C05444=1060.033,39.015,-71.744,171.703,28.984,155.388
C05445=1060.027,38.766,-71.728,171.703,28.981,155.388
C05446=1060.021,38.516,-71.712,171.701,28.979,155.387
C05447=1060.015,38.267,-71.695,171.699,28.976,155.387
C05448=1060.009,38.018,-71.679,171.698,28.973,155.387
C05449=1060.003,37.768,-71.663,171.696,28.971,155.386
C05450=1059.997,37.518,-71.646,171.695,28.968,155.386
C05451=1059.991,37.269,-71.630,171.693,28.966,155.386
C05452=1059.985,37.020,-71.614,171.692,28.963,155.385
C05453=1059.979,36.770,-71.598,171.690,28.961,155.385
C05454=1059.973,36.521,-71.583,171.688,28.959,155.385
C05455=1059.967,36.271,-71.566,171.688,28.956,155.384
C05456=1059.961,36.022,-71.550,171.686,28.954,155.384
C05457=1059.955,35.773,-71.534,171.684,28.951,155.383
C05458=1059.949,35.523,-71.518,171.683,28.949,155.383
C05459=1059.942,35.274,-71.502,171.681,28.946,155.383
C05460=1059.936,35.024,-71.485,171.680,28.944,155.382
C05461=1059.930,34.775,-71.469,171.679,28.941,155.382
C05462=1059.924,34.526,-71.453,171.677,28.939,155.382
C05463=1059.918,34.276,-71.437,171.675,28.936,155.381
C05464=1059.911,34.027,-71.422,171.674,28.933,155.381
C05465=1059.905,33.777,-71.405,171.673,28.931,155.381
C05466=1059.900,33.528,-71.389,171.671,28.929,155.380
C05467=1059.894,33.278,-71.373,171.670,28.927,155.380
C05468=1059.888,33.029,-71.357,171.668,28.924,155.380
C05469=1059.881,32.779,-71.342,171.666,28.922,155.379
C05470=1059.875,32.530,-71.325,171.666,28.919,155.379
C05471=1059.869,32.281,-71.309,171.664,28.916,155.379
C05472=1059.863,32.031,-71.293,171.662,28.914,155.378
C05473=1059.857,31.782,-71.277,171.661,28.911,155.378
C05474=1059.851,31.532,-71.262,171.659,28.909,155.378
C05475=1059.845,31.283,-71.245,171.658,28.906,155.377
C05476=1059.839,31.034,-71.229,171.657,28.904,155.377
C05477=1059.832,30.785,-71.213,171.655,28.901,155.377
C05478=1059.827,30.535,-71.198,171.653,28.899,155.376
C05479=1059.820,30.251,-71.179,171.652,28.896,155.376
C05480=1059.813,29.965,-71.162,171.650,28.893,155.375
C05481=1059.806,29.681,-71.143,171.649,28.890,155.375
C05482=1059.799,29.396,-71.125,171.647,28.888,155.375
C05483=1059.794,29.146,-71.108,171.645,28.885,155.374
C05484=1059.787,28.897,-71.093,171.644,28.883,155.374
C05485=1059.781,28.647,-71.077,171.642,28.880,155.374
C05486=1059.775,28.398,-71.061,171.641,28.878,155.373
C05487=1059.769,28.148,-71.046,171.640,28.876,155.373
C05488=1059.763,27.899,-71.030,171.638,28.873,155.373
C05489=1059.756,27.650,-71.014,171.636,28.871,155.372
C05490=1059.751,27.400,-70.999,171.635,28.868,155.372
C05491=1059.745,27.151,-70.982,171.634,28.866,155.372
C05492=1059.738,26.901,-70.967,171.632,28.863,155.371
C05493=1059.732,26.652,-70.951,171.631,28.861,155.371
C05494=1059.726,26.402,-70.935,171.629,28.858,155.371
C05495=1059.721,26.153,-70.920,171.627,28.856,155.370
C05496=1059.714,25.904,-70.905,171.626,28.853,155.370
C05497=1059.708,25.654,-70.889,171.625,28.851,155.370
C05498=1059.702,25.405,-70.873,171.623,28.848,155.369
C05499=1059.696,25.156,-70.857,171.622,28.846,155.369
C05500=1059.690,24.906,-70.842,171.620,28.843,155.368
C05501=1059.683,24.657,-70.826,171.618,28.841,155.368
C05502=1059.678,24.407,-70.810,171.618,28.838,155.368
C05503=1059.671,24.158,-70.795,171.616,28.836,155.367
C05504=1059.665,23.908,-70.779,171.614,28.833,155.367
C05505=1059.659,23.659,-70.764,171.613,28.831,155.367
C05506=1059.653,23.409,-70.748,171.611,28.829,155.367
C05507=1059.646,23.160,-70.732,171.609,28.826,155.366
C05508=1059.641,22.910,-70.717,171.608,28.824,155.366
C05509=1059.634,22.661,-70.702,171.607,28.822,155.365
C05510=1059.629,22.412,-70.686,171.605,28.819,155.365
C05511=1059.622,22.162,-70.670,171.604,28.817,155.365
C05512=1059.617,21.913,-70.655,171.602,28.814,155.365
C05513=1059.610,21.663,-70.639,171.601,28.812,155.364
C05514=1059.604,21.414,-70.624,171.599,28.810,155.364
C05515=1059.598,21.164,-70.607,171.598,28.807,155.363
C05516=1059.592,20.914,-70.592,171.596,28.805,155.363
C05517=1059.587,20.665,-70.577,171.595,28.802,155.363
C05518=1059.580,20.416,-70.562,171.593,28.800,155.362
C05519=1059.574,20.166,-70.546,171.592,28.797,155.362
C05520=1059.568,19.917,-70.530,171.590,28.795,155.362
C05521=1059.561,19.668,-70.515,171.589,28.793,155.362
C05522=1059.556,19.418,-70.500,171.587,28.790,155.361
C05523=1059.549,19.169,-70.484,171.585,28.788,155.361
C05524=1059.543,18.920,-70.470,171.584,28.785,155.360
C05525=1059.538,18.670,-70.454,171.583,28.783,155.360
C05526=1059.531,18.421,-70.438,171.581,28.781,155.360
C05527=1059.525,18.171,-70.423,171.580,28.778,155.359
C05528=1059.519,17.921,-70.408,171.578,28.776,155.359
C05529=1059.512,17.672,-70.392,171.577,28.773,155.359
C05530=1059.507,17.423,-70.377,171.576,28.771,155.359
C05531=1059.501,17.173,-70.362,171.574,28.769,155.358
C05532=1059.494,16.924,-70.346,171.572,28.766,155.358
C05533=1059.488,16.674,-70.331,171.571,28.764,155.358
C05534=1059.482,16.424,-70.316,171.569,28.761,155.357
C05535=1059.477,16.176,-70.300,171.567,28.759,155.357
C05536=1059.470,15.926,-70.285,171.567,28.757,155.357
C05537=1059.464,15.676,-70.270,171.565,28.754,155.356
C05538=1059.458,15.426,-70.255,171.563,28.752,155.356
C05539=1059.452,15.177,-70.239,171.562,28.749,155.356
C05540=1059.446,14.928,-70.224,171.560,28.747,155.355
C05541=1059.440,14.678,-70.209,171.558,28.744,155.355
C05542=1059.434,14.429,-70.194,171.558,28.742,155.355
C05543=1059.427,14.146,-70.176,171.555,28.739,155.354
C05544=1059.419,13.861,-70.160,171.554,28.737,155.354
C05545=1059.412,13.579,-70.142,171.552,28.734,155.354
C05546=1059.405,13.295,-70.125,171.550,28.731,155.353
C05547=1059.399,13.046,-70.110,171.549,28.729,155.353
C05548=1059.393,12.796,-70.095,171.547,28.727,155.353
C05549=1059.386,12.546,-70.080,171.546,28.725,155.352
C05550=1059.381,12.297,-70.065,171.545,28.722,155.352
C05551=1059.375,12.048,-70.050,171.543,28.720,155.352
C05552=1059.369,11.798,-70.035,171.541,28.717,155.351
C05553=1059.362,11.549,-70.019,171.540,28.715,155.351
C05554=1059.356,11.300,-70.005,171.538,28.712,155.351
C05555=1059.350,11.050,-69.990,171.537,28.710,155.350
C05556=1059.343,10.801,-69.975,171.536,28.708,155.350
C05557=1059.337,10.551,-69.960,171.534,28.705,155.350
C05558=1059.331,10.301,-69.945,171.532,28.703,155.349
C05559=1059.325,10.052,-69.930,171.531,28.701,155.349
C05560=1059.319,9.802,-69.915,171.529,28.699,155.349
C05561=1059.313,9.553,-69.900,171.527,28.696,155.349
C05562=1059.306,9.303,-69.885,171.527,28.694,155.348
C05563=1059.301,9.054,-69.870,171.525,28.692,155.348
C05564=1059.294,8.804,-69.855,171.523,28.689,155.348
C05565=1059.288,8.555,-69.840,171.522,28.687,155.347
C05566=1059.282,8.306,-69.826,171.520,28.684,155.347
C05567=1059.276,8.056,-69.811,171.518,28.682,155.347
C05568=1059.269,7.806,-69.796,171.516,28.680,155.347
C05569=1059.264,7.556,-69.780,171.516,28.677,155.346
C05570=1059.258,7.308,-69.766,171.514,28.675,155.346
C05571=1059.251,7.058,-69.751,171.512,28.673,155.346
C05572=1059.245,6.808,-69.736,171.511,28.671,155.345
C05573=1059.239,6.559,-69.721,171.509,28.668,155.345
C05574=1059.233,6.310,-69.706,171.507,28.666,155.345
C05575=1059.226,6.060,-69.691,171.506,28.664,155.344
C05576=1059.221,5.811,-69.677,171.505,28.662,155.344
C05577=1059.214,5.561,-69.662,171.503,28.659,155.344
C05578=1059.208,5.312,-69.647,171.502,28.656,155.343
C05579=1059.202,5.063,-69.632,171.500,28.654,155.343
C05580=1059.196,4.813,-69.617,171.498,28.652,155.343
C05581=1059.189,4.563,-69.602,171.497,28.649,155.342
C05582=1059.184,4.314,-69.588,171.495,28.647,155.342
C05583=1059.178,4.064,-69.573,171.494,28.645,155.342
C05584=1059.172,3.814,-69.558,171.493,28.643,155.342
C05585=1059.166,3.565,-69.544,171.491,28.640,155.341
C05586=1059.160,3.316,-69.529,171.489,28.638,155.341
C05587=1059.153,3.066,-69.514,171.488,28.636,155.341
C05588=1059.148,2.817,-69.499,171.486,28.633,155.340
C05589=1059.141,2.567,-69.484,171.484,28.631,155.340
C05590=1059.136,2.318,-69.470,171.484,28.629,155.340
C05591=1059.129,2.068,-69.455,171.482,28.626,155.339
C05592=1059.123,1.818,-69.440,171.480,28.624,155.339
C05593=1059.117,1.569,-69.426,171.479,28.621,155.339
C05594=1059.111,1.320,-69.411,171.477,28.619,155.338
C05595=1059.105,1.070,-69.397,171.475,28.617,155.338
C05596=1059.099,0.821,-69.382,171.474,28.615,155.338
C05597=1059.093,0.572,-69.367,171.473,28.612,155.338
C05598=1059.087,0.322,-69.353,171.471,28.610,155.337
C05599=1059.080,0.072,-69.338,171.470,28.608,155.337
C05600=1059.075,-0.177,-69.324,171.468,28.605,155.337
C05601=1059.068,-0.427,-69.309,171.466,28.603,155.336
C05602=1059.063,-0.676,-69.294,171.465,28.600,155.336
C05603=1059.056,-0.926,-69.279,171.463,28.598,155.336
C05604=1059.051,-1.175,-69.265,171.461,28.596,155.336
C05605=1059.044,-1.425,-69.250,171.461,28.593,155.335
C05606=1059.039,-1.674,-69.236,171.459,28.591,155.335
C05607=1059.032,-1.956,-69.219,171.457,28.589,155.335
C05608=1059.025,-2.237,-69.203,171.455,28.586,155.334
C05609=1059.018,-2.519,-69.187,171.453,28.583,155.334
C05610=1059.012,-2.801,-69.170,171.452,28.581,155.334
C05611=1059.006,-3.050,-69.155,171.450,28.578,155.333
C05612=1059.000,-3.299,-69.141,171.449,28.576,155.333
C05613=1058.993,-3.549,-69.127,171.448,28.574,155.333
C05614=1058.987,-3.798,-69.113,171.446,28.572,155.332
C05615=1058.981,-4.048,-69.098,171.444,28.569,155.332
C05616=1058.975,-4.298,-69.083,171.443,28.567,155.332
C05617=1058.968,-4.547,-69.069,171.441,28.565,155.331
C05618=1058.962,-4.797,-69.055,171.439,28.563,155.331
C05619=1058.956,-5.046,-69.041,171.438,28.560,155.331
C05620=1058.950,-5.296,-69.027,171.436,28.558,155.331
C05621=1058.944,-5.545,-69.012,171.435,28.556,155.330
C05622=1058.937,-5.794,-68.997,171.433,28.554,155.330
C05623=1058.932,-6.044,-68.984,171.432,28.552,155.330
C05624=1058.925,-6.293,-68.969,171.430,28.550,155.330
C05625=1058.919,-6.543,-68.955,171.428,28.547,155.329
C05626=1058.913,-6.793,-68.940,171.427,28.545,155.329
C05627=1058.906,-7.043,-68.927,171.425,28.543,155.329
C05628=1058.900,-7.291,-68.912,171.424,28.540,155.328
C05629=1058.894,-7.542,-68.898,171.422,28.538,155.328
C05630=1058.888,-7.790,-68.884,171.420,28.536,155.328
C05631=1058.882,-8.041,-68.870,171.419,28.534,155.328
C05632=1058.876,-8.290,-68.855,171.418,28.531,155.327
C05633=1058.870,-8.540,-68.841,171.416,28.529,155.327
C05634=1058.863,-8.789,-68.827,171.414,28.527,155.327
C05635=1058.858,-9.038,-68.813,171.413,28.525,155.326
C05636=1058.851,-9.288,-68.798,171.411,28.522,155.326
C05637=1058.845,-9.537,-68.785,171.409,28.520,155.326
C05638=1058.839,-9.787,-68.770,171.408,28.518,155.326
C05639=1058.833,-10.036,-68.756,171.406,28.516,155.325
C05640=1058.827,-10.286,-68.742,171.405,28.514,155.325
C05641=1058.821,-10.535,-68.728,171.404,28.512,155.325
C05642=1058.815,-10.786,-68.714,171.402,28.509,155.325
C05643=1058.808,-11.034,-68.700,171.400,28.507,155.324
C05644=1058.802,-11.284,-68.685,171.399,28.505,155.324
C05645=1058.797,-11.534,-68.672,171.397,28.503,155.324
C05646=1058.790,-11.783,-68.658,171.395,28.500,155.323
C05647=1058.784,-12.033,-68.643,171.394,28.498,155.323
C05648=1058.779,-12.282,-68.630,171.392,28.496,155.323
C05649=1058.771,-12.532,-68.615,171.390,28.494,155.323
C05650=1058.766,-12.781,-68.601,171.389,28.492,155.322
C05651=1058.760,-13.031,-68.588,171.388,28.490,155.322
C05652=1058.753,-13.280,-68.573,171.386,28.487,155.322
C05653=1058.748,-13.530,-68.559,171.385,28.485,155.322
C05654=1058.741,-13.780,-68.546,171.383,28.483,155.321
C05655=1058.735,-14.029,-68.531,171.381,28.481,155.321
C05656=1058.730,-14.278,-68.517,171.380,28.478,155.321
C05657=1058.723,-14.528,-68.504,171.378,28.476,155.320
C05658=1058.717,-14.777,-68.489,171.376,28.474,155.320
C05659=1058.711,-15.027,-68.476,171.375,28.472,155.320
C05660=1058.705,-15.277,-68.461,171.373,28.469,155.320
C05661=1058.699,-15.526,-68.448,171.371,28.467,155.319
C05662=1058.692,-15.776,-68.433,171.371,28.465,155.319
C05663=1058.686,-16.025,-68.420,171.369,28.464,155.319
C05664=1058.681,-16.275,-68.406,171.367,28.461,155.319
C05665=1058.674,-16.525,-68.392,171.365,28.459,155.318
C05666=1058.668,-16.774,-68.379,171.364,28.457,155.318
C05667=1058.661,-17.024,-68.364,171.362,28.455,155.318
C05668=1058.655,-17.273,-68.351,171.360,28.452,155.318
C05669=1058.650,-17.522,-68.337,171.359,28.450,155.317
C05670=1058.643,-17.772,-68.323,171.357,28.449,155.317
C05671=1058.636,-18.052,-68.307,171.355,28.446,155.317
C05672=1058.629,-18.332,-68.293,171.354,28.443,155.316
C05673=1058.622,-18.612,-68.277,171.352,28.441,155.316
C05674=1058.615,-18.892,-68.262,171.350,28.439,155.316
C05675=1058.609,-19.141,-68.248,171.349,28.437,155.316
C05676=1058.603,-19.391,-68.234,171.347,28.435,155.315
C05677=1058.596,-19.640,-68.220,171.345,28.432,155.315
C05678=1058.590,-19.889,-68.207,171.344,28.430,155.315
C05679=1058.584,-20.140,-68.193,171.342,28.428,155.315
C05680=1058.578,-20.389,-68.179,171.340,28.426,155.314
C05681=1058.573,-20.639,-68.166,171.339,28.424,155.314
C05682=1058.566,-20.889,-68.152,171.337,28.422,155.314
C05683=1058.559,-21.138,-68.139,171.335,28.419,155.314
C05684=1058.554,-21.387,-68.125,171.334,28.418,155.314
C05685=1058.548,-21.637,-68.112,171.332,28.416,155.313
C05686=1058.542,-21.887,-68.097,171.330,28.413,155.313
C05687=1058.535,-22.136,-68.084,171.329,28.411,155.313
C05688=1058.529,-22.385,-68.071,171.328,28.409,155.312
C05689=1058.523,-22.636,-68.057,171.326,28.407,155.312
C05690=1058.517,-22.885,-68.043,171.324,28.405,155.312
C05691=1058.511,-23.134,-68.030,171.323,28.403,155.312
C05692=1058.505,-23.384,-68.016,171.321,28.401,155.311
C05693=1058.498,-23.634,-68.003,171.319,28.399,155.311
C05694=1058.492,-23.883,-67.989,171.318,28.396,155.311
C05695=1058.487,-24.133,-67.975,171.316,28.395,155.311
C05696=1058.481,-24.382,-67.962,171.314,28.392,155.310
C05697=1058.474,-24.632,-67.948,171.313,28.390,155.310
C05698=1058.468,-24.881,-67.935,171.311,28.388,155.310
C05699=1058.462,-25.131,-67.921,171.309,28.386,155.310
C05700=1058.456,-25.380,-67.908,171.308,28.384,155.310
C05701=1058.450,-25.630,-67.894,171.306,28.382,155.309
C05702=1058.444,-25.880,-67.881,171.304,28.380,155.309
C05703=1058.437,-26.129,-67.867,171.303,28.377,155.309
C05704=1058.432,-26.378,-67.853,171.301,28.376,155.309
C05705=1058.426,-26.628,-67.840,171.300,28.374,155.308
C05706=1058.419,-26.878,-67.827,171.299,28.371,155.308
C05707=1058.414,-27.128,-67.813,171.297,28.369,155.308
C05708=1058.407,-27.377,-67.800,171.295,28.368,155.308
C05709=1058.401,-27.626,-67.787,171.294,28.365,155.307
C05710=1058.394,-27.876,-67.773,171.292,28.364,155.307
C05711=1058.388,-28.126,-67.760,171.290,28.361,155.307
C05712=1058.382,-28.375,-67.747,171.288,28.359,155.307
C05713=1058.376,-28.625,-67.734,171.287,28.358,155.306
C05714=1058.369,-28.875,-67.720,171.285,28.355,155.306
C05715=1058.363,-29.124,-67.707,171.283,28.353,155.306
C05716=1058.358,-29.373,-67.693,171.282,28.351,155.306
C05717=1058.351,-29.623,-67.680,171.280,28.349,155.306
C05718=1058.345,-29.873,-67.668,171.278,28.348,155.305
C05719=1058.339,-30.123,-67.654,171.277,28.345,155.305
C05720=1058.332,-30.372,-67.641,171.275,28.343,155.305
C05721=1058.326,-30.621,-67.627,171.273,28.341,155.305
C05722=1058.320,-30.870,-67.614,171.272,28.339,155.304
C05723=1058.314,-31.120,-67.602,171.270,28.337,155.304
C05724=1058.308,-31.370,-67.588,171.268,28.335,155.304
C05725=1058.301,-31.619,-67.575,171.266,28.333,155.304
C05726=1058.296,-31.870,-67.561,171.265,28.331,155.304
C05727=1058.290,-32.119,-67.548,171.263,28.329,155.303
C05728=1058.283,-32.368,-67.535,171.261,28.327,155.303
C05729=1058.277,-32.617,-67.522,171.260,28.325,155.303
C05730=1058.271,-32.867,-67.509,171.259,28.323,155.303
C05731=1058.265,-33.117,-67.495,171.257,28.322,155.302
C05732=1058.258,-33.367,-67.482,171.256,28.319,155.302
C05733=1058.252,-33.616,-67.470,171.254,28.318,155.302
C05734=1058.246,-33.866,-67.456,171.252,28.315,155.302
C05735=1058.240,-34.145,-67.442,171.250,28.313,155.302
C05736=1058.233,-34.424,-67.427,171.248,28.311,155.301
C05737=1058.226,-34.703,-67.413,171.246,28.308,155.301
C05738=1058.218,-34.982,-67.398,171.245,28.307,155.301
C05739=1058.212,-35.232,-67.385,171.243,28.305,155.301
C05740=1058.206,-35.482,-67.372,171.241,28.302,155.300
C05741=1058.200,-35.731,-67.359,171.239,28.301,155.300
C05742=1058.194,-35.981,-67.346,171.238,28.298,155.300
C05743=1058.188,-36.230,-67.333,171.236,28.297,155.300
C05744=1058.182,-36.480,-67.320,171.234,28.295,155.300
C05745=1058.177,-36.729,-67.306,171.233,28.293,155.299
C05746=1058.171,-36.979,-67.294,171.231,28.291,155.299
C05747=1058.164,-37.229,-67.280,171.229,28.289,155.299
C05748=1058.159,-37.478,-67.268,171.228,28.287,155.299
C05749=1058.152,-37.728,-67.255,171.226,28.285,155.298
C05750=1058.146,-37.978,-67.242,171.224,28.283,155.298
C05751=1058.140,-38.227,-67.229,171.223,28.281,155.298
C05752=1058.134,-38.477,-67.216,171.221,28.279,155.298
C05753=1058.128,-38.726,-67.203,171.219,28.277,155.298
C05754=1058.121,-38.976,-67.191,171.217,28.275,155.297
C05755=1058.115,-39.226,-67.177,171.216,28.273,155.297
C05756=1058.109,-39.475,-67.165,171.214,28.271,155.297
C05757=1058.102,-39.725,-67.152,171.212,28.270,155.297
C05758=1058.097,-39.975,-67.139,171.211,28.267,155.297
C05759=1058.090,-40.224,-67.126,171.209,28.266,155.296
C05760=1058.084,-40.473,-67.114,171.207,28.264,155.296
C05761=1058.077,-40.723,-67.100,171.206,28.262,155.296
C05762=1058.072,-40.973,-67.088,171.204,28.260,155.296
C05763=1058.066,-41.222,-67.075,171.202,28.258,155.296
C05764=1058.059,-41.472,-67.062,171.200,28.256,155.295
C05765=1058.053,-41.721,-67.050,171.199,28.254,155.295
C05766=1058.047,-41.970,-67.037,171.197,28.253,155.295
C05767=1058.041,-42.220,-67.024,171.195,28.251,155.295
C05768=1058.035,-42.470,-67.012,171.194,28.249,155.295
C05769=1058.029,-42.720,-66.998,171.192,28.247,155.295
C05770=1058.022,-42.969,-66.987,171.190,28.245,155.294
C05771=1058.016,-43.219,-66.974,171.188,28.243,155.294
C05772=1058.010,-43.468,-66.961,171.187,28.241,155.294
C05773=1058.004,-43.718,-66.948,171.185,28.239,155.294
C05774=1057.998,-43.968,-66.936,171.183,28.238,155.294
C05775=1057.991,-44.217,-66.923,171.182,28.236,155.293
C05776=1057.985,-44.467,-66.910,171.180,28.234,155.293
C05777=1057.979,-44.717,-66.898,171.178,28.232,155.293
C05778=1057.973,-44.966,-66.885,171.176,28.230,155.293
C05779=1057.966,-45.216,-66.873,171.175,28.228,155.293
C05780=1057.960,-45.465,-66.860,171.173,28.227,155.293
C05781=1057.955,-45.715,-66.847,171.171,28.225,155.292
C05782=1057.948,-45.965,-66.834,171.170,28.223,155.292
C05783=1057.942,-46.214,-66.822,171.168,28.221,155.292
C05784=1057.936,-46.464,-66.810,171.166,28.219,155.292
C05785=1057.930,-46.714,-66.797,171.165,28.217,155.292
C05786=1057.924,-46.963,-66.784,171.163,28.216,155.291
C05787=1057.917,-47.213,-66.772,171.161,28.214,155.291
C05788=1057.911,-47.463,-66.759,171.159,28.212,155.291
C05789=1057.906,-47.712,-66.747,171.158,28.210,155.291
C05790=1057.900,-47.961,-66.734,171.156,28.208,155.291
C05791=1057.893,-48.211,-66.722,171.154,28.207,155.291
C05792=1057.887,-48.461,-66.709,171.153,28.204,155.290
C05793=1057.881,-48.710,-66.697,171.151,28.203,155.290
C05794=1057.875,-48.960,-66.684,171.149,28.201,155.290
C05795=1057.869,-49.210,-66.672,171.147,28.199,155.290
C05796=1057.862,-49.459,-66.659,171.146,28.197,155.290
C05797=1057.856,-49.709,-66.646,171.144,28.196,155.289
C05798=1057.851,-49.958,-66.634,171.142,28.194,155.289
C05799=1057.843,-50.238,-66.620,171.141,28.192,155.289
C05800=1057.836,-50.518,-66.607,171.139,28.190,155.289
C05801=1057.830,-50.797,-66.593,171.136,28.187,155.289
C05802=1057.823,-51.077,-66.579,171.134,28.186,155.289
C05803=1057.816,-51.326,-66.568,171.133,28.184,155.288
C05804=1057.810,-51.576,-66.555,171.131,28.182,155.288
C05805=1057.804,-51.825,-66.542,171.129,28.181,155.288
C05806=1057.798,-52.075,-66.530,171.128,28.179,155.288
C05807=1057.791,-52.325,-66.518,171.126,28.178,155.288
C05808=1057.784,-52.574,-66.506,171.124,28.176,155.288
C05809=1057.778,-52.824,-66.493,171.122,28.174,155.287
C05810=1057.772,-53.074,-66.481,171.121,28.173,155.287
C05811=1057.766,-53.323,-66.469,171.119,28.171,155.287
C05812=1057.759,-53.573,-66.457,171.117,28.169,155.287
C05813=1057.753,-53.822,-66.445,171.115,28.168,155.287
C05814=1057.747,-54.072,-66.433,171.114,28.166,155.287
C05815=1057.741,-54.321,-66.421,171.112,28.164,155.287
C05816=1057.735,-54.571,-66.408,171.110,28.163,155.286
C05817=1057.728,-54.821,-66.396,171.109,28.161,155.286
C05818=1057.721,-55.070,-66.384,171.107,28.159,155.286
C05819=1057.716,-55.320,-66.372,171.105,28.158,155.286
C05820=1057.710,-55.570,-66.361,171.103,28.156,155.286
C05821=1057.704,-55.820,-66.348,171.102,28.154,155.286
C05822=1057.697,-56.069,-66.336,171.099,28.152,155.286
C05823=1057.691,-56.319,-66.324,171.097,28.151,155.285
C05824=1057.685,-56.569,-66.312,171.095,28.149,155.285
C05825=1057.678,-56.818,-66.300,171.094,28.147,155.285
C05826=1057.671,-57.068,-66.288,171.092,28.146,155.285
C05827=1057.666,-57.317,-66.276,171.090,28.144,155.285
C05828=1057.659,-57.567,-66.264,171.089,28.142,155.285
C05829=1057.654,-57.816,-66.251,171.087,28.141,155.285
C05830=1057.647,-58.067,-66.240,171.085,28.139,155.284
C05831=1057.641,-58.316,-66.228,171.083,28.137,155.284
C05832=1057.635,-58.565,-66.216,171.082,28.136,155.284
C05833=1057.629,-58.815,-66.204,171.080,28.134,155.284
C05834=1057.622,-59.065,-66.192,171.078,28.132,155.284
C05835=1057.616,-59.314,-66.179,171.076,28.131,155.284
C05836=1057.610,-59.564,-66.168,171.075,28.130,155.284
C05837=1057.604,-59.814,-66.156,171.073,28.128,155.284
C05838=1057.598,-60.063,-66.144,171.071,28.126,155.283
C05839=1057.591,-60.313,-66.132,171.069,28.125,155.283
C05840=1057.584,-60.563,-66.120,171.068,28.123,155.283
C05841=1057.579,-60.812,-66.109,171.066,28.121,155.283
C05842=1057.573,-61.062,-66.097,171.064,28.120,155.283
C05843=1057.566,-61.311,-66.085,171.062,28.118,155.283
C05844=1057.561,-61.561,-66.072,171.061,28.116,155.282
C05845=1057.554,-61.811,-66.061,171.059,28.115,155.282
C05846=1057.548,-62.060,-66.049,171.056,28.113,155.282
C05847=1057.542,-62.310,-66.037,171.055,28.112,155.282
C05848=1057.536,-62.559,-66.025,171.053,28.110,155.282
C05849=1057.530,-62.809,-66.014,171.051,28.108,155.282
C05850=1057.524,-63.059,-66.001,171.049,28.107,155.282
C05851=1057.518,-63.308,-65.990,171.048,28.105,155.282
C05852=1057.511,-63.558,-65.978,171.046,28.103,155.281
C05853=1057.505,-63.808,-65.966,171.044,28.102,155.281
C05854=1057.499,-64.058,-65.954,171.042,28.101,155.281
C05855=1057.493,-64.307,-65.942,171.041,28.099,155.281
C05856=1057.486,-64.557,-65.931,171.039,28.097,155.281
C05857=1057.480,-64.807,-65.919,171.037,28.096,155.281
C05858=1057.475,-65.056,-65.908,171.035,28.094,155.281
C05859=1057.468,-65.306,-65.896,171.034,28.092,155.281
C05860=1057.462,-65.556,-65.883,171.032,28.091,155.281
C05861=1057.456,-65.805,-65.872,171.030,28.090,155.280
C05862=1057.450,-66.055,-65.860,171.028,28.088,155.280
C05863=1057.440,-66.445,-65.842,171.025,28.085,155.280
C05864=1057.431,-66.836,-65.823,171.022,28.083,155.280
C05865=1057.422,-67.226,-65.805,171.020,28.080,155.280
C05866=1057.412,-67.617,-65.787,171.017,28.078,155.280
C05867=1057.406,-67.867,-65.776,171.015,28.077,155.279
C05868=1057.399,-68.116,-65.764,171.014,28.075,155.279
C05869=1057.394,-68.366,-65.752,171.012,28.073,155.279
C05870=1057.388,-68.616,-65.740,171.010,28.072,155.279
C05871=1057.381,-68.866,-65.729,171.008,28.071,155.279
C05872=1057.375,-69.115,-65.717,171.006,28.069,155.279
C05873=1057.370,-69.365,-65.706,171.004,28.067,155.279
C05874=1057.364,-69.614,-65.694,171.002,28.065,155.279
C05875=1057.357,-69.864,-65.683,171.000,28.064,155.278
C05876=1057.351,-70.113,-65.671,170.999,28.063,155.278
C05877=1057.346,-70.364,-65.659,170.997,28.061,155.278
C05878=1057.339,-70.613,-65.647,170.995,28.059,155.278
C05879=1057.333,-70.863,-65.637,170.993,28.058,155.278
C05880=1057.327,-71.112,-65.625,170.992,28.057,155.278
C05881=1057.322,-71.362,-65.613,170.990,28.055,155.278
C05882=1057.315,-71.612,-65.601,170.988,28.053,155.278
C05883=1057.309,-71.861,-65.590,170.986,28.052,155.278
C05884=1057.303,-72.111,-65.579,170.985,28.050,155.277
C05885=1057.297,-72.360,-65.567,170.983,28.049,155.277
C05886=1057.291,-72.611,-65.556,170.981,28.048,155.277
C05887=1057.285,-72.860,-65.544,170.979,28.046,155.277
C05888=1057.279,-73.110,-65.533,170.978,28.044,155.277
C05889=1057.273,-73.359,-65.522,170.975,28.042,155.277
C05890=1057.266,-73.609,-65.510,170.973,28.041,155.277
C05891=1057.261,-73.859,-65.498,170.971,28.040,155.277
C05892=1057.255,-74.108,-65.487,170.970,28.039,155.277
C05893=1057.249,-74.358,-65.476,170.968,28.037,155.276
C05894=1057.243,-74.608,-65.464,170.966,28.035,155.276
C05895=1057.237,-74.857,-65.453,170.964,28.034,155.276
C05896=1057.230,-75.107,-65.442,170.963,28.033,155.276
C05897=1057.224,-75.357,-65.430,170.961,28.031,155.276
C05898=1057.218,-75.607,-65.419,170.959,28.030,155.276
C05899=1057.212,-75.856,-65.407,170.957,28.029,155.276
C05900=1057.206,-76.106,-65.397,170.956,28.027,155.276
C05901=1057.199,-76.356,-65.385,170.954,28.026,155.276
C05902=1057.193,-76.605,-65.374,170.952,28.024,155.276
C05903=1057.186,-76.855,-65.363,170.949,28.023,155.276
C05904=1057.181,-77.104,-65.352,170.947,28.021,155.276
C05905=1057.174,-77.354,-65.341,170.946,28.020,155.275
C05906=1057.168,-77.603,-65.329,170.944,28.019,155.275
C05907=1057.162,-77.853,-65.318,170.942,28.018,155.275
C05908=1057.156,-78.103,-65.307,170.940,28.016,155.275
C05909=1057.150,-78.353,-65.296,170.939,28.015,155.275
C05910=1057.144,-78.603,-65.285,170.937,28.014,155.275
C05911=1057.134,-78.992,-65.268,170.934,28.011,155.275
C05912=1057.125,-79.382,-65.250,170.931,28.009,155.275
C05913=1057.115,-79.771,-65.233,170.928,28.007,155.275
C05914=1057.105,-80.161,-65.215,170.925,28.005,155.275
C05915=1057.100,-80.411,-65.204,170.924,28.004,155.274
C05916=1057.093,-80.661,-65.193,170.922,28.002,155.274
C05917=1057.087,-80.910,-65.183,170.920,28.001,155.274
C05918=1057.080,-81.159,-65.171,170.918,28.000,155.274
C05919=1057.074,-81.409,-65.160,170.915,27.998,155.274
C05920=1057.069,-81.658,-65.149,170.914,27.997,155.274
C05921=1057.062,-81.908,-65.139,170.912,27.996,155.274
C05922=1057.056,-82.158,-65.128,170.910,27.995,155.274
C05923=1057.048,-82.441,-65.116,170.908,27.994,155.274
C05924=1057.041,-82.724,-65.103,170.905,27.992,155.274
C05925=1057.035,-83.007,-65.090,170.904,27.991,155.274
C05926=1057.027,-83.290,-65.078,170.902,27.989,155.274
C05927=1057.021,-83.540,-65.067,170.900,27.988,155.274
C05928=1057.015,-83.789,-65.056,170.897,27.986,155.274
C05929=1057.008,-84.039,-65.045,170.896,27.985,155.274
C05930=1057.003,-84.289,-65.034,170.894,27.984,155.274
C05931=1056.996,-84.539,-65.023,170.892,27.983,155.274
C05932=1056.990,-84.788,-65.013,170.890,27.982,155.274
C05933=1056.984,-85.038,-65.002,170.888,27.981,155.274
C05934=1056.978,-85.288,-64.991,170.887,27.979,155.273
C05935=1056.971,-85.537,-64.980,170.885,27.978,155.273
C05936=1056.965,-85.787,-64.969,170.883,27.977,155.273
C05937=1056.959,-86.037,-64.958,170.881,27.976,155.273
C05938=1056.953,-86.286,-64.948,170.880,27.975,155.273
C05939=1056.947,-86.537,-64.937,170.877,27.973,155.273
C05940=1056.941,-86.786,-64.927,170.875,27.972,155.273
C05941=1056.934,-87.035,-64.916,170.873,27.971,155.273
C05942=1056.928,-87.286,-64.905,170.871,27.970,155.273
C05943=1056.922,-87.535,-64.894,170.870,27.969,155.273
C05944=1056.916,-87.784,-64.884,170.868,27.967,155.273
C05945=1056.909,-88.035,-64.873,170.866,27.966,155.273
C05946=1056.904,-88.284,-64.862,170.864,27.965,155.273
C05947=1056.897,-88.533,-64.851,170.862,27.964,155.273
C05948=1056.891,-88.783,-64.840,170.861,27.963,155.273
C05949=1056.885,-89.033,-64.829,170.858,27.962,155.273
C05950=1056.879,-89.283,-64.820,170.856,27.961,155.273
C05951=1056.873,-89.533,-64.809,170.854,27.959,155.273
C05952=1056.867,-89.782,-64.798,170.852,27.958,155.273
C05953=1056.860,-90.032,-64.787,170.851,27.957,155.273
C05954=1056.854,-90.282,-64.776,170.849,27.956,155.273
C05955=1056.848,-90.531,-64.765,170.847,27.955,155.273
C05956=1056.842,-90.781,-64.756,170.845,27.953,155.273
C05957=1056.836,-91.030,-64.745,170.843,27.952,155.273
C05958=1056.829,-91.280,-64.734,170.842,27.951,155.273
C05959=1056.824,-91.530,-64.723,170.839,27.950,155.273
C05960=1056.818,-91.779,-64.712,170.837,27.949,155.273
C05961=1056.811,-92.030,-64.702,170.835,27.948,155.273
C05962=1056.805,-92.279,-64.692,170.833,27.947,155.272
C05963=1056.800,-92.529,-64.681,170.832,27.945,155.272
C05964=1056.793,-92.778,-64.670,170.830,27.944,155.272
C05965=1056.787,-93.029,-64.660,170.828,27.943,155.272
C05966=1056.781,-93.278,-64.650,170.826,27.942,155.272
C05967=1056.775,-93.527,-64.639,170.824,27.941,155.272
C05968=1056.769,-93.777,-64.628,170.823,27.940,155.272
C05969=1056.762,-94.027,-64.618,170.820,27.938,155.272
C05970=1056.757,-94.277,-64.607,170.818,27.937,155.272
C05971=1056.750,-94.526,-64.597,170.816,27.936,155.272
C05972=1056.745,-94.776,-64.587,170.814,27.935,155.272
C05973=1056.739,-95.026,-64.576,170.813,27.934,155.272
C05974=1056.732,-95.276,-64.565,170.811,27.933,155.272
C05975=1056.726,-95.526,-64.555,170.809,27.932,155.272
C05976=1056.720,-95.775,-64.545,170.807,27.931,155.272
C05977=1056.714,-96.024,-64.534,170.805,27.930,155.272
C05978=1056.709,-96.274,-64.524,170.804,27.929,155.272
C05979=1056.702,-96.524,-64.513,170.801,27.927,155.272
C05980=1056.696,-96.774,-64.502,170.799,27.926,155.272
C05981=1056.690,-97.024,-64.492,170.797,27.925,155.272
C05982=1056.684,-97.273,-64.482,170.795,27.924,155.272
C05983=1056.678,-97.523,-64.472,170.793,27.924,155.272
C05984=1056.672,-97.772,-64.461,170.792,27.923,155.272
C05985=1056.665,-98.022,-64.451,170.790,27.922,155.272
C05986=1056.660,-98.272,-64.440,170.788,27.920,155.272
C05987=1056.652,-98.557,-64.429,170.785,27.919,155.272
C05988=1056.645,-98.843,-64.417,170.783,27.918,155.272
C05989=1056.638,-99.128,-64.405,170.781,27.917,155.272
C05990=1056.631,-99.413,-64.394,170.779,27.916,155.272
C05991=1056.625,-99.663,-64.384,170.777,27.915,155.272
C05992=1056.619,-99.913,-64.373,170.775,27.914,155.272
C05993=1056.612,-100.163,-64.363,170.773,27.913,155.272
C05994=1056.606,-100.412,-64.353,170.772,27.912,155.272
C05995=1056.601,-100.662,-64.342,170.769,27.911,155.272
C05996=1056.594,-100.912,-64.333,170.767,27.910,155.272
C05997=1056.588,-101.161,-64.323,170.765,27.909,155.272
C05998=1056.582,-101.412,-64.312,170.763,27.908,155.272
C05999=1056.575,-101.661,-64.302,170.761,27.907,155.272
C06000=1056.569,-101.911,-64.292,170.760,27.906,155.272
C06001=1056.563,-102.160,-64.281,170.758,27.905,155.272
C06002=1056.557,-102.410,-64.272,170.756,27.905,155.272
C06003=1056.551,-102.660,-64.262,170.754,27.904,155.272
C06004=1056.545,-102.909,-64.251,170.751,27.902,155.272
C06005=1056.539,-103.159,-64.242,170.749,27.902,155.272
C06006=1056.532,-103.409,-64.231,170.748,27.901,155.272
C06007=1056.526,-103.659,-64.221,170.746,27.900,155.272
C06008=1056.520,-103.908,-64.211,170.744,27.899,155.272
C06009=1056.514,-104.158,-64.201,170.742,27.898,155.272
C06010=1056.508,-104.408,-64.191,170.740,27.897,155.272
C06011=1056.502,-104.657,-64.181,170.738,27.897,155.272
C06012=1056.496,-104.907,-64.171,170.737,27.896,155.272
C06013=1056.490,-105.157,-64.161,170.734,27.894,155.272
C06014=1056.484,-105.406,-64.151,170.732,27.894,155.272
C06015=1056.478,-105.656,-64.141,170.730,27.893,155.272
C06016=1056.472,-105.906,-64.131,170.728,27.892,155.272
C06017=1056.465,-106.155,-64.121,170.726,27.891,155.272
C06018=1056.459,-106.406,-64.111,170.725,27.890,155.272
C06019=1056.453,-106.656,-64.101,170.723,27.890,155.272
C06020=1056.447,-106.905,-64.091,170.721,27.889,155.272
C06021=1056.440,-107.155,-64.081,170.718,27.887,155.272
C06022=1056.434,-107.404,-64.072,170.716,27.887,155.272
C06023=1056.429,-107.655,-64.061,170.714,27.886,155.272
C06024=1056.422,-107.904,-64.051,170.713,27.885,155.273
C06025=1056.416,-108.154,-64.042,170.711,27.884,155.273
C06026=1056.410,-108.403,-64.032,170.709,27.884,155.273
C06027=1056.404,-108.653,-64.023,170.707,27.883,155.273
C06028=1056.397,-108.902,-64.012,170.705,27.882,155.273
C06029=1056.391,-109.152,-64.003,170.703,27.881,155.273
C06030=1056.386,-109.402,-63.992,170.700,27.880,155.273
C06031=1056.380,-109.652,-63.983,170.699,27.880,155.273
C06032=1056.373,-109.901,-63.973,170.697,27.879,155.273
C06033=1056.367,-110.151,-63.963,170.695,27.878,155.273
C06034=1056.361,-110.401,-63.954,170.693,27.877,155.273
C06035=1056.355,-110.651,-63.944,170.691,27.877,155.273
C06036=1056.348,-110.900,-63.934,170.689,27.876,155.273
C06037=1056.342,-111.150,-63.925,170.687,27.875,155.273
C06038=1056.336,-111.399,-63.915,170.685,27.874,155.273
C06039=1056.330,-111.649,-63.905,170.683,27.873,155.273
C06040=1056.324,-111.899,-63.895,170.681,27.873,155.273
C06041=1056.318,-112.149,-63.885,170.679,27.872,155.273
C06042=1056.312,-112.399,-63.876,170.677,27.871,155.273
C06043=1056.306,-112.649,-63.866,170.675,27.870,155.273
C06044=1056.299,-112.898,-63.857,170.673,27.870,155.273
C06045=1056.293,-113.148,-63.847,170.672,27.869,155.273
C06046=1056.287,-113.397,-63.837,170.669,27.868,155.273
C06047=1056.281,-113.647,-63.827,170.667,27.867,155.274
C06048=1056.274,-113.897,-63.818,170.665,27.867,155.274
C06049=1056.268,-114.147,-63.808,170.663,27.866,155.274
C06050=1056.262,-114.397,-63.798,170.661,27.865,155.274
C06051=1056.255,-114.680,-63.787,170.659,27.865,155.274
C06052=1056.248,-114.964,-63.776,170.657,27.864,155.274
C06053=1056.241,-115.249,-63.766,170.655,27.863,155.274
C06054=1056.234,-115.532,-63.755,170.652,27.862,155.274
C06055=1056.228,-115.782,-63.745,170.650,27.861,155.274
C06056=1056.222,-116.032,-63.736,170.648,27.861,155.274
C06057=1056.216,-116.282,-63.726,170.646,27.860,155.274
C06058=1056.210,-116.531,-63.717,170.644,27.860,155.274
C06059=1056.204,-116.781,-63.707,170.643,27.859,155.274
C06060=1056.198,-117.031,-63.698,170.641,27.858,155.274
C06061=1056.192,-117.280,-63.688,170.638,27.858,155.275
C06062=1056.186,-117.530,-63.679,170.636,27.857,155.275
C06063=1056.179,-117.780,-63.669,170.634,27.857,155.275
C06064=1056.173,-118.030,-63.660,170.632,27.856,155.275
C06065=1056.166,-118.279,-63.651,170.630,27.855,155.275
C06066=1056.160,-118.529,-63.641,170.628,27.855,155.275
C06067=1056.154,-118.779,-63.631,170.627,27.854,155.275
C06068=1056.148,-119.029,-63.622,170.625,27.854,155.275
C06069=1056.142,-119.278,-63.613,170.622,27.853,155.275
C06070=1056.136,-119.528,-63.604,170.620,27.852,155.275
C06071=1056.130,-119.778,-63.594,170.618,27.851,155.275
C06072=1056.124,-120.028,-63.585,170.616,27.851,155.275
C06073=1056.118,-120.277,-63.575,170.614,27.850,155.275
C06074=1056.112,-120.527,-63.566,170.612,27.850,155.275
C06075=1056.105,-120.777,-63.557,170.611,27.849,155.276
C06076=1056.099,-121.026,-63.547,170.609,27.849,155.276
C06077=1056.093,-121.276,-63.538,170.606,27.848,155.276
C06078=1056.087,-121.526,-63.529,170.604,27.847,155.276
C06079=1056.081,-121.776,-63.519,170.602,27.847,155.276
C06080=1056.075,-122.026,-63.510,170.600,27.846,155.276
C06081=1056.069,-122.275,-63.500,170.598,27.846,155.276
C06082=1056.062,-122.525,-63.491,170.596,27.845,155.276
C06083=1056.056,-122.775,-63.483,170.594,27.845,155.276
C06084=1056.050,-123.024,-63.473,170.593,27.844,155.276
C06085=1056.044,-123.274,-63.464,170.590,27.844,155.276
C06086=1056.038,-123.524,-63.454,170.588,27.843,155.277
C06087=1056.032,-123.774,-63.445,170.586,27.843,155.277
C06088=1056.026,-124.024,-63.436,170.584,27.842,155.277
C06089=1056.020,-124.273,-63.427,170.582,27.842,155.277
C06090=1056.013,-124.523,-63.418,170.580,27.841,155.277
C06091=1056.007,-124.773,-63.408,170.578,27.841,155.277
C06092=1056.001,-125.023,-63.399,170.576,27.840,155.277
C06093=1055.995,-125.272,-63.391,170.574,27.840,155.277
C06094=1055.989,-125.522,-63.381,170.572,27.839,155.277
C06095=1055.983,-125.772,-63.372,170.570,27.839,155.277
C06096=1055.976,-126.022,-63.363,170.568,27.838,155.277
C06097=1055.970,-126.271,-63.354,170.566,27.838,155.278
C06098=1055.965,-126.521,-63.345,170.564,27.838,155.278
C06099=1055.959,-126.771,-63.335,170.562,27.837,155.278
C06100=1055.952,-127.020,-63.327,170.559,27.837,155.278
C06101=1055.946,-127.271,-63.318,170.557,27.836,155.278
C06102=1055.940,-127.521,-63.308,170.555,27.836,155.278
C06103=1055.933,-127.769,-63.300,170.554,27.835,155.278
C06104=1055.928,-128.020,-63.290,170.552,27.835,155.278
C06105=1055.924,-128.270,-63.280,170.550,27.833,155.278
C06106=1055.921,-128.520,-63.269,170.548,27.831,155.278
C06107=1055.920,-128.770,-63.258,170.547,27.829,155.278
C06108=1055.919,-129.021,-63.245,170.545,27.826,155.277
C06109=1055.919,-129.271,-63.232,170.545,27.823,155.277
C06110=1055.922,-129.522,-63.218,170.543,27.819,155.276
C06111=1055.925,-129.773,-63.205,170.542,27.814,155.276
C06112=1055.929,-130.024,-63.190,170.542,27.809,155.275
C06113=1055.935,-130.275,-63.174,170.542,27.803,155.274
C06114=1055.942,-130.525,-63.157,170.541,27.797,155.273
C06115=1055.569,-130.548,-63.365,170.493,27.963,155.306
C06116=1055.562,-130.298,-63.382,170.493,27.968,155.307
C06117=1055.557,-130.047,-63.397,170.494,27.974,155.308
C06118=1055.552,-129.796,-63.412,170.495,27.979,155.309
C06119=1055.549,-129.544,-63.426,170.496,27.984,155.310
C06120=1055.546,-129.295,-63.440,170.496,27.988,155.310
C06121=1055.546,-129.044,-63.453,170.498,27.992,155.311
C06122=1055.546,-128.794,-63.465,170.499,27.994,155.311
C06123=1055.548,-128.543,-63.477,170.501,27.997,155.311
C06124=1055.551,-128.293,-63.487,170.502,27.999,155.311
C06125=1055.555,-128.043,-63.497,170.504,28.000,155.312
C06126=1055.560,-127.793,-63.508,170.506,28.001,155.312
C06127=1055.566,-127.543,-63.516,170.508,28.001,155.311
C06128=1055.572,-127.294,-63.525,170.510,28.001,155.311
C06129=1055.579,-127.044,-63.535,170.512,28.002,155.311
C06130=1055.585,-126.794,-63.543,170.514,28.002,155.311
C06131=1055.591,-126.544,-63.553,170.516,28.003,155.311
C06132=1055.597,-126.295,-63.562,170.519,28.004,155.311
C06133=1055.603,-126.045,-63.571,170.520,28.004,155.311
C06134=1055.609,-125.795,-63.580,170.522,28.005,155.311
C06135=1055.616,-125.545,-63.589,170.524,28.005,155.311
C06136=1055.622,-125.295,-63.598,170.526,28.005,155.310
C06137=1055.627,-125.046,-63.607,170.528,28.005,155.310
C06138=1055.634,-124.796,-63.617,170.530,28.006,155.310
C06139=1055.640,-124.547,-63.626,170.533,28.007,155.310
C06140=1055.646,-124.296,-63.634,170.535,28.007,155.310
C06141=1055.652,-124.046,-63.644,170.537,28.007,155.310
C06142=1055.658,-123.797,-63.653,170.539,28.008,155.310
C06143=1055.664,-123.547,-63.663,170.541,28.008,155.310
C06144=1055.671,-123.297,-63.671,170.542,28.009,155.310
C06145=1055.677,-123.048,-63.681,170.544,28.009,155.310
C06146=1055.683,-122.798,-63.690,170.546,28.010,155.309
C06147=1055.689,-122.548,-63.700,170.549,28.010,155.309
C06148=1055.695,-122.299,-63.709,170.551,28.011,155.309
C06149=1055.701,-122.048,-63.718,170.553,28.011,155.309
C06150=1055.707,-121.799,-63.727,170.555,28.013,155.309
C06151=1055.714,-121.549,-63.736,170.557,28.013,155.309
C06152=1055.720,-121.299,-63.746,170.558,28.013,155.309
C06153=1055.726,-121.050,-63.756,170.560,28.014,155.309
C06154=1055.732,-120.800,-63.765,170.563,28.015,155.309
C06155=1055.738,-120.550,-63.774,170.565,28.015,155.309
C06156=1055.744,-120.300,-63.783,170.567,28.016,155.309
C06157=1055.750,-120.050,-63.793,170.569,28.016,155.309
C06158=1055.756,-119.801,-63.802,170.571,28.016,155.308
C06159=1055.763,-119.551,-63.811,170.573,28.017,155.308
C06160=1055.769,-119.301,-63.821,170.575,28.018,155.308
C06161=1055.775,-119.052,-63.830,170.576,28.019,155.308
C06162=1055.781,-118.802,-63.840,170.579,28.019,155.308
C06163=1055.787,-118.553,-63.849,170.581,28.020,155.308
C06164=1055.793,-118.302,-63.858,170.583,28.020,155.308
C06165=1055.799,-118.052,-63.868,170.585,28.021,155.308
C06166=1055.805,-117.803,-63.877,170.587,28.022,155.308
C06167=1055.812,-117.553,-63.887,170.589,28.022,155.308
C06168=1055.818,-117.303,-63.896,170.591,28.023,155.308
C06169=1055.824,-117.053,-63.906,170.593,28.023,155.308
C06170=1055.830,-116.803,-63.915,170.595,28.024,155.308
C06171=1055.836,-116.554,-63.925,170.597,28.025,155.308
C06172=1055.842,-116.304,-63.935,170.599,28.025,155.307
C06173=1055.848,-116.055,-63.944,170.601,28.026,155.307
C06174=1055.855,-115.805,-63.953,170.603,28.026,155.307
C06175=1055.861,-115.556,-63.962,170.605,28.027,155.307
C06176=1055.869,-115.271,-63.974,170.608,28.028,155.307
C06177=1055.875,-114.988,-63.985,170.609,28.029,155.307
C06178=1055.882,-114.704,-63.996,170.612,28.029,155.307
C06179=1055.889,-114.420,-64.006,170.614,28.030,155.307
C06180=1055.895,-114.170,-64.015,170.616,28.031,155.307
C06181=1055.901,-113.920,-64.025,170.618,28.031,155.307
C06182=1055.908,-113.671,-64.035,170.620,28.032,155.307
C06183=1055.914,-113.421,-64.045,170.622,28.033,155.307
C06184=1055.919,-113.171,-64.055,170.625,28.033,155.307
C06185=1055.925,-112.921,-64.065,170.626,28.035,155.307
C06186=1055.932,-112.671,-64.074,170.628,28.035,155.307
C06187=1055.938,-112.422,-64.084,170.630,28.036,155.307
C06188=1055.944,-112.172,-64.093,170.632,28.037,155.306
C06189=1055.950,-111.922,-64.103,170.634,28.037,155.306
C06190=1055.956,-111.672,-64.112,170.636,28.038,155.306
C06191=1055.963,-111.423,-64.123,170.638,28.039,155.306
C06192=1055.969,-111.173,-64.132,170.640,28.040,155.306
C06193=1055.975,-110.923,-64.142,170.642,28.040,155.306
C06194=1055.981,-110.674,-64.151,170.644,28.041,155.306
C06195=1055.987,-110.424,-64.161,170.646,28.042,155.306
C06196=1055.993,-110.174,-64.171,170.648,28.042,155.306
C06197=1055.999,-109.925,-64.181,170.650,28.043,155.306
C06198=1056.006,-109.675,-64.191,170.652,28.044,155.306
C06199=1056.012,-109.425,-64.200,170.654,28.045,155.306
C06200=1056.018,-109.175,-64.210,170.656,28.046,155.306
C06201=1056.024,-108.925,-64.220,170.658,28.046,155.306
C06202=1056.031,-108.676,-64.230,170.660,28.047,155.306
C06203=1056.036,-108.426,-64.240,170.662,28.048,155.306
C06204=1056.042,-108.176,-64.250,170.664,28.049,155.306
C06205=1056.048,-107.927,-64.259,170.666,28.049,155.306
C06206=1056.055,-107.677,-64.269,170.667,28.050,155.306
C06207=1056.061,-107.428,-64.279,170.670,28.051,155.306
C06208=1056.068,-107.177,-64.289,170.672,28.052,155.306
C06209=1056.073,-106.928,-64.300,170.674,28.053,155.306
C06210=1056.080,-106.678,-64.309,170.676,28.054,155.306
C06211=1056.086,-106.428,-64.319,170.678,28.055,155.306
C06212=1056.092,-106.178,-64.329,170.679,28.055,155.306
C06213=1056.098,-105.929,-64.339,170.681,28.056,155.306
C06214=1056.104,-105.679,-64.349,170.683,28.057,155.305
C06215=1056.110,-105.429,-64.359,170.686,28.058,155.305
C06216=1056.117,-105.180,-64.369,170.688,28.059,155.305
C06217=1056.122,-104.930,-64.379,170.690,28.060,155.305
C06218=1056.128,-104.680,-64.389,170.691,28.061,155.305
C06219=1056.135,-104.431,-64.399,170.693,28.061,155.305
C06220=1056.141,-104.181,-64.408,170.695,28.062,155.305
C06221=1056.147,-103.932,-64.419,170.697,28.063,155.305
C06222=1056.153,-103.681,-64.429,170.699,28.064,155.305
C06223=1056.159,-103.431,-64.439,170.702,28.065,155.305
C06224=1056.165,-103.182,-64.450,170.703,28.066,155.305
C06225=1056.171,-102.932,-64.459,170.705,28.067,155.305
C06226=1056.178,-102.683,-64.470,170.707,28.068,155.305
C06227=1056.183,-102.433,-64.480,170.709,28.069,155.305
C06228=1056.190,-102.183,-64.490,170.711,28.069,155.305
C06229=1056.196,-101.934,-64.500,170.713,28.070,155.305
C06230=1056.202,-101.683,-64.510,170.715,28.071,155.305
C06231=1056.208,-101.434,-64.520,170.716,28.072,155.305
C06232=1056.215,-101.184,-64.530,170.719,28.073,155.305
C06233=1056.220,-100.934,-64.541,170.721,28.074,155.305
C06234=1056.227,-100.685,-64.550,170.723,28.075,155.305
C06235=1056.233,-100.435,-64.561,170.725,28.076,155.305
C06236=1056.238,-100.185,-64.571,170.727,28.077,155.305
C06237=1056.246,-99.935,-64.581,170.728,28.078,155.305
C06238=1056.252,-99.686,-64.591,170.730,28.079,155.305
C06239=1056.257,-99.436,-64.602,170.732,28.080,155.305
C06240=1056.264,-99.150,-64.613,170.735,28.081,155.305
C06241=1056.272,-98.866,-64.625,170.737,28.082,155.305
C06242=1056.279,-98.580,-64.636,170.739,28.083,155.305
C06243=1056.286,-98.294,-64.649,170.741,28.084,155.305
C06244=1056.292,-98.045,-64.658,170.743,28.085,155.305
C06245=1056.298,-97.795,-64.669,170.745,28.086,155.305
C06246=1056.304,-97.545,-64.679,170.747,28.087,155.305
C06247=1056.311,-97.295,-64.690,170.750,28.088,155.305
C06248=1056.317,-97.046,-64.700,170.751,28.089,155.305
C06249=1056.323,-96.796,-64.710,170.753,28.090,155.305
C06250=1056.329,-96.547,-64.721,170.755,28.091,155.305
C06251=1056.335,-96.297,-64.732,170.757,28.092,155.305
C06252=1056.340,-96.047,-64.742,170.759,28.093,155.305
C06253=1056.347,-95.797,-64.752,170.760,28.094,155.305
C06254=1056.353,-95.548,-64.763,170.762,28.096,155.305
C06255=1056.359,-95.298,-64.773,170.764,28.097,155.305
C06256=1056.365,-95.048,-64.784,170.767,28.098,155.305
C06257=1056.371,-94.799,-64.795,170.769,28.099,155.305
C06258=1056.377,-94.548,-64.805,170.770,28.100,155.305
C06259=1056.383,-94.299,-64.815,170.772,28.101,155.305
C06260=1056.390,-94.050,-64.826,170.774,28.102,155.305
C06261=1056.395,-93.800,-64.836,170.776,28.103,155.305
C06262=1056.401,-93.550,-64.847,170.778,28.104,155.305
C06263=1056.408,-93.300,-64.857,170.780,28.105,155.305
C06264=1056.414,-93.051,-64.868,170.781,28.106,155.306
C06265=1056.420,-92.801,-64.878,170.783,28.108,155.306
C06266=1056.426,-92.552,-64.889,170.786,28.109,155.306
C06267=1056.432,-92.301,-64.900,170.788,28.110,155.306
C06268=1056.438,-92.052,-64.910,170.790,28.111,155.306
C06269=1056.444,-91.802,-64.920,170.791,28.112,155.306
C06270=1056.450,-91.553,-64.931,170.793,28.113,155.306
C06271=1056.457,-91.303,-64.942,170.795,28.114,155.306
C06272=1056.462,-91.053,-64.953,170.797,28.115,155.306
C06273=1056.469,-90.804,-64.963,170.799,28.117,155.306
C06274=1056.475,-90.553,-64.974,170.800,28.118,155.306
C06275=1056.481,-90.304,-64.984,170.802,28.119,155.306
C06276=1056.487,-90.055,-64.995,170.805,28.120,155.306
C06277=1056.493,-89.805,-65.006,170.807,28.121,155.306
C06278=1056.499,-89.555,-65.017,170.809,28.122,155.306
C06279=1056.506,-89.306,-65.027,170.810,28.124,155.306
C06280=1056.511,-89.056,-65.037,170.812,28.125,155.306
C06281=1056.517,-88.805,-65.049,170.814,28.126,155.306
C06282=1056.524,-88.556,-65.059,170.816,28.127,155.306
C06283=1056.530,-88.307,-65.070,170.818,28.128,155.306
C06284=1056.536,-88.057,-65.081,170.819,28.129,155.306
C06285=1056.543,-87.807,-65.091,170.822,28.131,155.306
C06286=1056.548,-87.558,-65.102,170.824,28.132,155.306
C06287=1056.555,-87.308,-65.113,170.826,28.133,155.306
C06288=1056.561,-87.059,-65.124,170.828,28.134,155.306
C06289=1056.567,-86.809,-65.135,170.829,28.135,155.306
C06290=1056.573,-86.559,-65.146,170.831,28.136,155.306
C06291=1056.579,-86.309,-65.155,170.833,28.138,155.306
C06292=1056.586,-86.059,-65.167,170.835,28.139,155.307
C06293=1056.591,-85.809,-65.177,170.837,28.140,155.307
C06294=1056.598,-85.560,-65.188,170.838,28.141,155.307
C06295=1056.604,-85.310,-65.199,170.841,28.142,155.307
C06296=1056.610,-85.060,-65.210,170.843,28.144,155.307
C06297=1056.617,-84.811,-65.221,170.845,28.145,155.307
C06298=1056.623,-84.561,-65.231,170.847,28.146,155.307
C06299=1056.629,-84.312,-65.242,170.848,28.147,155.307
C06300=1056.636,-84.062,-65.253,170.850,28.148,155.307
C06301=1056.641,-83.812,-65.264,170.852,28.150,155.307
C06302=1056.648,-83.562,-65.275,170.854,28.151,155.307
C06303=1056.653,-83.313,-65.286,170.856,28.152,155.307
C06304=1056.661,-83.030,-65.298,170.858,28.153,155.307
C06305=1056.668,-82.746,-65.311,170.860,28.155,155.307
C06306=1056.675,-82.464,-65.323,170.862,28.156,155.307
C06307=1056.682,-82.181,-65.336,170.865,28.158,155.307
C06308=1056.689,-81.931,-65.346,170.866,28.159,155.307
C06309=1056.695,-81.681,-65.357,170.868,28.160,155.307
C06310=1056.701,-81.431,-65.368,170.870,28.161,155.307
C06311=1056.707,-81.181,-65.379,170.872,28.163,155.308
C06312=1056.714,-80.932,-65.390,170.874,28.164,155.308
C06313=1056.720,-80.683,-65.402,170.875,28.165,155.308
C06314=1056.726,-80.433,-65.413,170.877,28.166,155.308
C06315=1056.732,-80.183,-65.424,170.880,28.168,155.308
C06316=1056.739,-79.933,-65.434,170.882,28.169,155.308
C06317=1056.745,-79.684,-65.445,170.884,28.170,155.308
C06318=1056.751,-79.433,-65.456,170.885,28.172,155.308
C06319=1056.757,-79.184,-65.467,170.887,28.173,155.308
C06320=1056.763,-78.934,-65.479,170.889,28.174,155.308
C06321=1056.769,-78.685,-65.490,170.891,28.176,155.308
C06322=1056.775,-78.435,-65.501,170.892,28.177,155.308
C06323=1056.781,-78.185,-65.512,170.894,28.178,155.308
C06324=1056.787,-77.936,-65.524,170.896,28.179,155.308
C06325=1056.794,-77.686,-65.535,170.898,28.181,155.308
C06326=1056.799,-77.437,-65.546,170.900,28.182,155.309
C06327=1056.806,-77.187,-65.557,170.902,28.184,155.309
C06328=1056.812,-76.937,-65.568,170.904,28.185,155.309
C06329=1056.818,-76.687,-65.580,170.906,28.187,155.309
C06330=1056.824,-76.438,-65.591,170.908,28.188,155.309
C06331=1056.830,-76.188,-65.602,170.909,28.189,155.309
C06332=1056.836,-75.939,-65.614,170.911,28.190,155.309
C06333=1056.843,-75.689,-65.624,170.913,28.192,155.309
C06334=1056.849,-75.440,-65.635,170.915,28.193,155.309
C06335=1056.855,-75.189,-65.647,170.916,28.195,155.309
C06336=1056.862,-74.940,-65.658,170.918,28.196,155.309
C06337=1056.868,-74.690,-65.669,170.920,28.198,155.309
C06338=1056.874,-74.440,-65.681,170.922,28.199,155.310
C06339=1056.880,-74.191,-65.692,170.924,28.200,155.310
C06340=1056.887,-73.941,-65.703,170.926,28.202,155.310
C06341=1056.892,-73.692,-65.716,170.928,28.203,155.310
C06342=1056.898,-73.442,-65.727,170.930,28.205,155.310
C06343=1056.904,-73.192,-65.738,170.932,28.206,155.310
C06344=1056.911,-72.943,-65.750,170.933,28.208,155.310
C06345=1056.916,-72.693,-65.761,170.935,28.209,155.310
C06346=1056.922,-72.443,-65.772,170.937,28.210,155.310
C06347=1056.928,-72.194,-65.784,170.939,28.212,155.310
C06348=1056.934,-71.944,-65.795,170.940,28.214,155.311
C06349=1056.940,-71.695,-65.807,170.942,28.215,155.311
C06350=1056.946,-71.444,-65.819,170.944,28.216,155.311
C06351=1056.952,-71.195,-65.830,170.946,28.218,155.311
C06352=1056.958,-70.945,-65.842,170.947,28.220,155.311
C06353=1056.965,-70.696,-65.854,170.949,28.221,155.311
C06354=1056.971,-70.446,-65.864,170.951,28.222,155.311
C06355=1056.977,-70.196,-65.877,170.954,28.224,155.311
C06356=1056.982,-69.947,-65.888,170.955,28.225,155.311
C06357=1056.989,-69.697,-65.900,170.957,28.227,155.312
C06358=1056.995,-69.448,-65.911,170.959,28.229,155.312
C06359=1057.001,-69.198,-65.923,170.961,28.230,155.312
C06360=1057.006,-68.948,-65.934,170.962,28.231,155.312
C06361=1057.013,-68.699,-65.946,170.964,28.233,155.312
C06362=1057.019,-68.448,-65.957,170.966,28.235,155.312
C06363=1057.025,-68.199,-65.969,170.968,28.236,155.312
C06364=1057.031,-67.949,-65.981,170.969,28.238,155.312
C06365=1057.037,-67.700,-65.992,170.971,28.239,155.312
C06366=1057.043,-67.450,-66.004,170.973,28.241,155.313
C06367=1057.049,-67.200,-66.016,170.975,28.243,155.313
C06368=1057.057,-66.919,-66.029,170.977,28.244,155.313
C06369=1057.062,-66.639,-66.042,170.979,28.246,155.313
C06370=1057.070,-66.358,-66.055,170.981,28.248,155.313
C06371=1057.076,-66.077,-66.069,170.983,28.249,155.313
C06372=1057.083,-65.827,-66.081,170.985,28.251,155.313
C06373=1057.089,-65.577,-66.092,170.987,28.253,155.314
C06374=1057.095,-65.328,-66.103,170.989,28.254,155.314
C06375=1057.101,-65.078,-66.115,170.991,28.256,155.314
C06376=1057.108,-64.828,-66.127,170.992,28.257,155.314
C06377=1057.114,-64.579,-66.139,170.994,28.259,155.314
C06378=1057.119,-64.329,-66.151,170.996,28.261,155.314
C06379=1057.126,-64.079,-66.163,170.998,28.262,155.314
C06380=1057.132,-63.830,-66.174,170.999,28.263,155.314
C06381=1057.139,-63.581,-66.186,171.001,28.265,155.314
C06382=1057.144,-63.330,-66.198,171.003,28.267,155.315
C06383=1057.150,-63.081,-66.210,171.005,28.268,155.315
C06384=1057.157,-62.832,-66.222,171.006,28.270,155.315
C06385=1057.162,-62.581,-66.233,171.008,28.272,155.315
C06386=1057.169,-62.332,-66.245,171.010,28.273,155.315
C06387=1057.175,-62.083,-66.257,171.012,28.274,155.315
C06388=1057.181,-61.833,-66.270,171.013,28.276,155.315
C06389=1057.187,-61.583,-66.281,171.015,28.278,155.316
C06390=1057.193,-61.334,-66.292,171.017,28.279,155.316
C06391=1057.199,-61.084,-66.305,171.019,28.281,155.316
C06392=1057.206,-60.834,-66.317,171.020,28.283,155.316
C06393=1057.212,-60.584,-66.328,171.023,28.285,155.316
C06394=1057.218,-60.335,-66.340,171.025,28.286,155.316
C06395=1057.224,-60.085,-66.352,171.027,28.287,155.316
C06396=1057.231,-59.836,-66.364,171.028,28.289,155.316
C06397=1057.237,-59.586,-66.377,171.030,28.291,155.317
C06398=1057.243,-59.337,-66.388,171.032,28.292,155.317
C06399=1057.249,-59.087,-66.400,171.034,28.294,155.317
C06400=1057.255,-58.837,-66.412,171.035,28.296,155.317
C06401=1057.262,-58.587,-66.424,171.037,28.297,155.317
C06402=1057.268,-58.338,-66.436,171.039,28.299,155.317
C06403=1057.274,-58.089,-66.448,171.040,28.300,155.317
C06404=1057.280,-57.839,-66.460,171.042,28.302,155.318
C06405=1057.286,-57.589,-66.472,171.044,28.304,155.318
C06406=1057.293,-57.339,-66.484,171.046,28.305,155.318
C06407=1057.299,-57.090,-66.496,171.047,28.307,155.318
C06408=1057.305,-56.840,-66.509,171.049,28.308,155.318
C06409=1057.311,-56.591,-66.520,171.051,28.310,155.318
C06410=1057.318,-56.341,-66.532,171.053,28.311,155.318
C06411=1057.324,-56.091,-66.545,171.054,28.313,155.319
C06412=1057.330,-55.842,-66.557,171.056,28.315,155.319
C06413=1057.336,-55.592,-66.569,171.058,28.316,155.319
C06414=1057.343,-55.342,-66.581,171.060,28.318,155.319
C06415=1057.349,-55.093,-66.593,171.061,28.320,155.319
C06416=1057.359,-54.686,-66.613,171.065,28.322,155.319
C06417=1057.369,-54.279,-66.633,171.068,28.326,155.320
C06418=1057.380,-53.873,-66.652,171.070,28.328,155.320
C06419=1057.390,-53.466,-66.672,171.074,28.331,155.320
C06420=1057.396,-53.217,-66.684,171.075,28.332,155.320
C06421=1057.402,-52.967,-66.696,171.077,28.334,155.320
C06422=1057.408,-52.717,-66.708,171.079,28.336,155.320
C06423=1057.415,-52.468,-66.720,171.081,28.337,155.321
C06424=1057.421,-52.218,-66.733,171.082,28.339,155.321
C06425=1057.428,-51.968,-66.745,171.084,28.341,155.321
C06426=1057.434,-51.719,-66.757,171.086,28.342,155.321
C06427=1057.440,-51.470,-66.770,171.088,28.344,155.321
C06428=1057.449,-51.097,-66.788,171.090,28.346,155.321
C06429=1057.459,-50.724,-66.806,171.093,28.349,155.322
C06430=1057.469,-50.353,-66.824,171.095,28.351,155.322
C06431=1057.478,-49.980,-66.843,171.098,28.354,155.322
C06432=1057.484,-49.730,-66.855,171.100,28.356,155.322
C06433=1057.490,-49.480,-66.868,171.101,28.358,155.323
C06434=1057.496,-49.231,-66.881,171.103,28.359,155.323
C06435=1057.502,-48.982,-66.893,171.105,28.362,155.323
C06436=1057.508,-48.732,-66.905,171.107,28.363,155.323
C06437=1057.514,-48.483,-66.918,171.108,28.365,155.323
C06438=1057.520,-48.233,-66.930,171.110,28.367,155.323
C06439=1057.526,-47.984,-66.943,171.112,28.369,155.324
C06440=1057.532,-47.734,-66.956,171.114,28.370,155.324
C06441=1057.538,-47.484,-66.968,171.115,28.372,155.324
C06442=1057.545,-47.234,-66.980,171.117,28.374,155.324
C06443=1057.551,-46.985,-66.993,171.119,28.376,155.324
C06444=1057.557,-46.735,-67.006,171.120,28.378,155.325
C06445=1057.563,-46.485,-67.018,171.122,28.379,155.325
C06446=1057.570,-46.236,-67.030,171.124,28.382,155.325
C06447=1057.576,-45.986,-67.043,171.126,28.383,155.325
C06448=1057.582,-45.737,-67.056,171.127,28.385,155.325
C06449=1057.588,-45.487,-67.069,171.129,28.387,155.325
C06450=1057.594,-45.238,-67.080,171.131,28.389,155.326
C06451=1057.600,-44.989,-67.094,171.132,28.390,155.326
C06452=1057.606,-44.739,-67.106,171.134,28.392,155.326
C06453=1057.612,-44.489,-67.119,171.136,28.394,155.326
C06454=1057.618,-44.239,-67.131,171.138,28.396,155.326
C06455=1057.625,-43.990,-67.144,171.139,28.398,155.326
C06456=1057.630,-43.740,-67.156,171.141,28.400,155.327
C06457=1057.636,-43.490,-67.169,171.143,28.402,155.327
C06458=1057.643,-43.241,-67.182,171.145,28.403,155.327
C06459=1057.649,-42.991,-67.194,171.146,28.405,155.327
C06460=1057.655,-42.742,-67.208,171.148,28.407,155.327
C06461=1057.661,-42.492,-67.220,171.150,28.409,155.328
C06462=1057.667,-42.242,-67.233,171.151,28.411,155.328
C06463=1057.674,-41.993,-67.246,171.153,28.413,155.328
C06464=1057.680,-41.744,-67.258,171.155,28.414,155.328
C06465=1057.686,-41.494,-67.270,171.156,28.416,155.328
C06466=1057.693,-41.244,-67.284,171.158,28.418,155.329
C06467=1057.699,-40.994,-67.297,171.160,28.420,155.329
C06468=1057.705,-40.745,-67.310,171.162,28.422,155.329
C06469=1057.711,-40.495,-67.322,171.163,28.424,155.329
C06470=1057.718,-40.246,-67.335,171.165,28.426,155.329
C06471=1057.724,-39.996,-67.348,171.167,28.428,155.330
C06472=1057.730,-39.747,-67.361,171.169,28.429,155.330
C06473=1057.736,-39.497,-67.373,171.170,28.431,155.330
C06474=1057.742,-39.247,-67.386,171.172,28.433,155.330
C06475=1057.749,-38.998,-67.399,171.174,28.435,155.330
C06476=1057.755,-38.748,-67.411,171.175,28.437,155.331
C06477=1057.761,-38.499,-67.425,171.177,28.439,155.331
C06478=1057.767,-38.249,-67.437,171.179,28.441,155.331
C06479=1057.773,-38.000,-67.450,171.181,28.443,155.331
C06480=1057.779,-37.750,-67.463,171.182,28.445,155.331
C06481=1057.785,-37.500,-67.476,171.184,28.446,155.332
C06482=1057.792,-37.250,-67.490,171.186,28.449,155.332
C06483=1057.798,-37.001,-67.502,171.187,28.450,155.332
C06484=1057.804,-36.751,-67.516,171.189,28.453,155.332
C06485=1057.810,-36.501,-67.528,171.191,28.454,155.332
C06486=1057.816,-36.252,-67.541,171.192,28.456,155.333
C06487=1057.821,-36.002,-67.555,171.194,28.458,155.333
C06488=1057.828,-35.753,-67.568,171.196,28.460,155.333
C06489=1057.834,-35.503,-67.581,171.198,28.462,155.333
C06490=1057.840,-35.254,-67.594,171.199,28.464,155.333
C06491=1057.846,-35.004,-67.607,171.201,28.466,155.334
C06492=1057.853,-34.725,-67.621,171.203,28.468,155.334
C06493=1057.860,-34.446,-67.636,171.204,28.470,155.334
C06494=1057.867,-34.166,-67.651,171.206,28.473,155.334
C06495=1057.873,-33.887,-67.665,171.208,28.475,155.335
C06496=1057.880,-33.638,-67.678,171.209,28.477,155.335
C06497=1057.886,-33.389,-67.692,171.211,28.479,155.335
C06498=1057.892,-33.139,-67.704,171.213,28.481,155.335
C06499=1057.899,-32.889,-67.718,171.215,28.483,155.336
C06500=1057.905,-32.639,-67.731,171.216,28.485,155.336
C06501=1057.911,-32.390,-67.744,171.218,28.486,155.336
C06502=1057.917,-32.140,-67.757,171.220,28.489,155.336
C06503=1057.923,-31.891,-67.770,171.221,28.491,155.336
C06504=1057.929,-31.641,-67.784,171.223,28.493,155.337
C06505=1057.935,-31.391,-67.797,171.225,28.495,155.337
C06506=1057.941,-31.142,-67.810,171.226,28.496,155.337
C06507=1057.948,-30.892,-67.824,171.228,28.499,155.337
C06508=1057.954,-30.643,-67.837,171.230,28.500,155.337
C06509=1057.960,-30.393,-67.849,171.232,28.502,155.338
C06510=1057.966,-30.143,-67.863,171.233,28.505,155.338
C06511=1057.973,-29.894,-67.876,171.235,28.506,155.338
C06512=1057.979,-29.645,-67.890,171.237,28.509,155.338
C06513=1057.985,-29.395,-67.903,171.238,28.510,155.339
C06514=1057.990,-29.145,-67.916,171.240,28.512,155.339
C06515=1057.997,-28.895,-67.930,171.242,28.515,155.339
C06516=1058.003,-28.646,-67.943,171.243,28.516,155.339
C06517=1058.010,-28.397,-67.956,171.245,28.519,155.340
C06518=1058.016,-28.147,-67.969,171.247,28.520,155.340
C06519=1058.022,-27.898,-67.982,171.248,28.522,155.340
C06520=1058.028,-27.648,-67.996,171.249,28.524,155.340
C06521=1058.035,-27.398,-68.009,171.251,28.526,155.340
C06522=1058.040,-27.149,-68.023,171.253,28.528,155.341
C06523=1058.047,-26.899,-68.036,171.254,28.531,155.341
C06524=1058.053,-26.650,-68.050,171.256,28.532,155.341
C06525=1058.059,-26.400,-68.063,171.258,28.534,155.341
C06526=1058.065,-26.151,-68.077,171.259,28.537,155.342
C06527=1058.071,-25.901,-68.089,171.261,28.539,155.342
C06528=1058.078,-25.651,-68.103,171.263,28.541,155.342
C06529=1058.083,-25.401,-68.117,171.265,28.543,155.342
C06530=1058.089,-25.152,-68.130,171.266,28.545,155.343
C06531=1058.095,-24.903,-68.143,171.268,28.547,155.343
C06532=1058.102,-24.652,-68.158,171.270,28.549,155.343
C06533=1058.108,-24.403,-68.171,171.271,28.551,155.343
C06534=1058.114,-24.154,-68.184,171.273,28.553,155.344
C06535=1058.119,-23.904,-68.198,171.275,28.556,155.344
C06536=1058.126,-23.654,-68.212,171.275,28.558,155.344
C06537=1058.133,-23.405,-68.225,171.277,28.559,155.344
C06538=1058.138,-23.156,-68.239,171.279,28.561,155.345
C06539=1058.144,-22.906,-68.252,171.281,28.564,155.345
C06540=1058.151,-22.656,-68.266,171.282,28.566,155.345
C06541=1058.156,-22.407,-68.280,171.284,28.568,155.345
C06542=1058.163,-22.158,-68.293,171.286,28.570,155.345
C06543=1058.168,-21.908,-68.307,171.287,28.572,155.346
C06544=1058.175,-21.658,-68.320,171.289,28.574,155.346
C06545=1058.181,-21.409,-68.334,171.291,28.576,155.346
C06546=1058.187,-21.159,-68.347,171.292,28.579,155.347
C06547=1058.194,-20.910,-68.362,171.294,28.580,155.347
C06548=1058.200,-20.661,-68.375,171.296,28.583,155.347
C06549=1058.205,-20.411,-68.389,171.297,28.585,155.347
C06550=1058.212,-20.161,-68.403,171.299,28.587,155.347
C06551=1058.218,-19.911,-68.416,171.300,28.589,155.348
C06552=1058.224,-19.662,-68.430,171.302,28.591,155.348
C06553=1058.231,-19.412,-68.443,171.303,28.593,155.348
C06554=1058.236,-19.163,-68.457,171.305,28.595,155.348
C06555=1058.243,-18.913,-68.470,171.307,28.597,155.349
C06556=1058.249,-18.634,-68.487,171.308,28.600,155.349
C06557=1058.257,-18.353,-68.502,171.310,28.602,155.349
C06558=1058.263,-18.073,-68.518,171.313,28.604,155.350
C06559=1058.271,-17.793,-68.533,171.314,28.607,155.350
C06560=1058.277,-17.544,-68.547,171.316,28.609,155.350
C06561=1058.283,-17.295,-68.560,171.318,28.611,155.350
C06562=1058.289,-17.045,-68.574,171.319,28.613,155.351
C06563=1058.295,-16.795,-68.588,171.320,28.615,155.351
C06564=1058.302,-16.545,-68.602,171.322,28.617,155.351
C06565=1058.307,-16.296,-68.616,171.323,28.620,155.351
C06566=1058.314,-16.047,-68.629,171.325,28.621,155.352
C06567=1058.320,-15.797,-68.643,171.327,28.623,155.352
C06568=1058.326,-15.547,-68.657,171.329,28.626,155.352
C06569=1058.333,-15.298,-68.671,171.330,28.628,155.352
C06570=1058.338,-15.049,-68.685,171.332,28.630,155.353
C06571=1058.345,-14.799,-68.699,171.334,28.632,155.353
C06572=1058.351,-14.549,-68.713,171.335,28.635,155.353
C06573=1058.357,-14.300,-68.727,171.337,28.637,155.353
C06574=1058.363,-14.050,-68.741,171.339,28.639,155.354
C06575=1058.369,-13.801,-68.755,171.339,28.641,155.354
C06576=1058.375,-13.552,-68.769,171.341,28.643,155.354
C06577=1058.381,-13.302,-68.783,171.343,28.645,155.355
C06578=1058.387,-13.052,-68.797,171.344,28.648,155.355
C06579=1058.394,-12.803,-68.811,171.346,28.650,155.355
C06580=1058.400,-12.553,-68.825,171.348,28.652,155.355
C06581=1058.405,-12.304,-68.839,171.349,28.654,155.356
C06582=1058.412,-12.054,-68.853,171.351,28.657,155.356
C06583=1058.418,-11.805,-68.867,171.353,28.659,155.356
C06584=1058.424,-11.554,-68.881,171.354,28.661,155.356
C06585=1058.430,-11.306,-68.895,171.355,28.663,155.357
C06586=1058.436,-11.055,-68.909,171.357,28.665,155.357
C06587=1058.442,-10.806,-68.924,171.359,28.667,155.357
C06588=1058.448,-10.557,-68.937,171.360,28.670,155.358
C06589=1058.454,-10.307,-68.952,171.362,28.672,155.358
C06590=1058.460,-10.058,-68.966,171.364,28.674,155.358
C06591=1058.467,-9.808,-68.980,171.365,28.676,155.358
C06592=1058.473,-9.559,-68.994,171.367,28.679,155.359
C06593=1058.479,-9.309,-69.009,171.369,28.681,155.359
C06594=1058.485,-9.060,-69.023,171.369,28.683,155.359
C06595=1058.491,-8.810,-69.037,171.371,28.685,155.360
C06596=1058.497,-8.561,-69.051,171.373,28.687,155.360
C06597=1058.504,-8.311,-69.065,171.374,28.689,155.360
C06598=1058.510,-8.062,-69.080,171.376,28.692,155.360
C06599=1058.516,-7.812,-69.094,171.378,28.694,155.361
C06600=1058.522,-7.563,-69.108,171.380,28.696,155.361
C06601=1058.528,-7.313,-69.122,171.381,28.698,155.361
C06602=1058.534,-7.064,-69.137,171.383,28.701,155.361
C06603=1058.540,-6.814,-69.151,171.385,28.703,155.362
C06604=1058.547,-6.565,-69.165,171.385,28.705,155.362
C06605=1058.553,-6.315,-69.179,171.387,28.707,155.362
C06606=1058.559,-6.066,-69.194,171.389,28.709,155.363
C06607=1058.566,-5.816,-69.207,171.390,28.711,155.363
C06608=1058.571,-5.567,-69.222,171.392,28.714,155.363
C06609=1058.578,-5.317,-69.237,171.394,28.716,155.363
C06610=1058.584,-5.067,-69.251,171.395,28.718,155.364
C06611=1058.590,-4.818,-69.265,171.397,28.720,155.364
C06612=1058.596,-4.568,-69.279,171.398,28.722,155.364
C06613=1058.602,-4.319,-69.294,171.400,28.725,155.364
C06614=1058.609,-4.070,-69.308,171.401,28.727,155.365
C06615=1058.615,-3.820,-69.322,171.403,28.729,155.365
C06616=1058.621,-3.570,-69.337,171.405,28.731,155.365
C06617=1058.627,-3.320,-69.351,171.406,28.733,155.366
C06618=1058.633,-3.071,-69.366,171.408,28.736,155.366
C06619=1058.639,-2.821,-69.381,171.410,28.738,155.366
C06620=1058.646,-2.540,-69.397,171.411,28.741,155.366
C06621=1058.653,-2.258,-69.413,171.413,28.743,155.367
C06622=1058.659,-1.977,-69.430,171.415,28.746,155.367
C06623=1058.667,-1.695,-69.446,171.416,28.748,155.368
C06624=1058.673,-1.446,-69.460,171.418,28.751,155.368
C06625=1058.679,-1.196,-69.475,171.419,28.754,155.368
C06626=1058.684,-0.947,-69.489,171.421,28.756,155.368
C06627=1058.691,-0.697,-69.504,171.423,28.758,155.369
C06628=1058.697,-0.448,-69.519,171.424,28.760,155.369
C06629=1058.703,-0.199,-69.534,171.425,28.762,155.369
C06630=1058.709,0.052,-69.548,171.427,28.765,155.370
C06631=1058.715,0.301,-69.562,171.429,28.767,155.370
C06632=1058.721,0.550,-69.577,171.430,28.769,155.370
C06633=1058.727,0.799,-69.592,171.432,28.772,155.371
C06634=1058.733,1.049,-69.607,171.434,28.774,155.371
C06635=1058.739,1.299,-69.621,171.434,28.776,155.371
C06636=1058.745,1.548,-69.636,171.436,28.779,155.371
C06637=1058.752,1.798,-69.651,171.438,28.781,155.372
C06638=1058.757,2.047,-69.666,171.439,28.783,155.372
C06639=1058.763,2.297,-69.681,171.441,28.786,155.372
C06640=1058.769,2.546,-69.695,171.443,28.788,155.373
C06641=1058.775,2.796,-69.709,171.444,28.790,155.373
C06642=1058.781,3.046,-69.724,171.445,28.792,155.373
C06643=1058.787,3.295,-69.739,171.447,28.795,155.374
C06644=1058.793,3.544,-69.754,171.448,28.797,155.374
C06645=1058.800,3.794,-69.769,171.450,28.799,155.374
C06646=1058.806,4.043,-69.783,171.452,28.802,155.374
C06647=1058.812,4.293,-69.798,171.453,28.804,155.375
C06648=1058.818,4.542,-69.813,171.455,28.807,155.375
C06649=1058.824,4.792,-69.827,171.456,28.809,155.375
C06650=1058.830,5.041,-69.842,171.458,28.811,155.376
C06651=1058.836,5.290,-69.857,171.459,28.813,155.376
C06652=1058.842,5.540,-69.872,171.461,28.816,155.376
C06653=1058.849,5.790,-69.887,171.463,28.818,155.377
C06654=1058.855,6.039,-69.902,171.464,28.820,155.377
C06655=1058.861,6.288,-69.916,171.466,28.823,155.377
C06656=1058.867,6.538,-69.932,171.467,28.825,155.378
C06657=1058.873,6.788,-69.947,171.468,28.827,155.378
C06658=1058.879,7.037,-69.961,171.470,28.830,155.378
C06659=1058.885,7.287,-69.976,171.472,28.832,155.378
C06660=1058.892,7.536,-69.991,171.473,28.835,155.379
C06661=1058.897,7.785,-70.006,171.475,28.837,155.379
C06662=1058.904,8.035,-70.021,171.476,28.839,155.379
C06663=1058.910,8.285,-70.036,171.477,28.841,155.380
C06664=1058.916,8.534,-70.051,171.479,28.844,155.380
C06665=1058.922,8.783,-70.065,171.481,28.846,155.380
C06666=1058.929,9.033,-70.080,171.482,28.848,155.381
C06667=1058.934,9.283,-70.096,171.484,28.850,155.381
C06668=1058.941,9.532,-70.111,171.486,28.853,155.381
C06669=1058.946,9.781,-70.125,171.487,28.855,155.382
C06670=1058.953,10.031,-70.140,171.488,28.857,155.382
C06671=1058.959,10.281,-70.155,171.490,28.860,155.382
C06672=1058.966,10.530,-70.170,171.492,28.862,155.382
C06673=1058.972,10.779,-70.185,171.493,28.865,155.383
C06674=1058.978,11.028,-70.200,171.495,28.867,155.383
C06675=1058.984,11.278,-70.215,171.496,28.869,155.383
C06676=1058.990,11.528,-70.231,171.497,28.871,155.384
C06677=1058.996,11.777,-70.245,171.499,28.874,155.384
C06678=1059.002,12.027,-70.260,171.501,28.876,155.384
C06679=1059.009,12.276,-70.275,171.502,28.878,155.385
C06680=1059.015,12.526,-70.290,171.504,28.880,155.385
C06681=1059.022,12.775,-70.306,171.505,28.883,155.385
C06682=1059.028,13.025,-70.321,171.506,28.885,155.386
C06683=1059.034,13.274,-70.335,171.508,28.887,155.386
C06684=1059.041,13.558,-70.353,171.510,28.890,155.386
C06685=1059.048,13.841,-70.370,171.511,28.893,155.387
C06686=1059.055,14.124,-70.387,171.513,28.895,155.387
C06687=1059.062,14.409,-70.405,171.516,28.898,155.387
C06688=1059.068,14.657,-70.419,171.516,28.900,155.388
C06689=1059.074,14.907,-70.435,171.518,28.903,155.388
C06690=1059.080,15.156,-70.450,171.520,28.905,155.388
C06691=1059.086,15.406,-70.465,171.521,28.908,155.389
C06692=1059.093,15.656,-70.480,171.523,28.910,155.389
C06693=1059.098,15.904,-70.496,171.525,28.912,155.389
C06694=1059.104,16.154,-70.511,171.525,28.915,155.390
C06695=1059.111,16.404,-70.526,171.527,28.917,155.390
C06696=1059.117,16.653,-70.542,171.529,28.919,155.390
C06697=1059.123,16.903,-70.557,171.530,28.922,155.390
C06698=1059.130,17.152,-70.572,171.532,28.924,155.391
C06699=1059.135,17.402,-70.587,171.533,28.927,155.391
C06700=1059.141,17.651,-70.603,171.535,28.929,155.391
C06701=1059.147,17.901,-70.619,171.536,28.931,155.392
C06702=1059.153,18.150,-70.634,171.538,28.934,155.392
C06703=1059.160,18.399,-70.649,171.540,28.936,155.392
C06704=1059.166,18.649,-70.665,171.541,28.939,155.393
C06705=1059.172,18.898,-70.680,171.542,28.941,155.393
C06706=1059.177,19.148,-70.696,171.544,28.943,155.393
C06707=1059.184,19.397,-70.711,171.545,28.946,155.394
C06708=1059.190,19.646,-70.726,171.547,28.948,155.394
C06709=1059.196,19.896,-70.742,171.549,28.951,155.394
C06710=1059.202,20.146,-70.757,171.550,28.953,155.395
C06711=1059.208,20.395,-70.773,171.551,28.955,155.395
C06712=1059.215,20.645,-70.788,171.553,28.958,155.395
C06713=1059.220,20.894,-70.804,171.554,28.960,155.396
C06714=1059.226,21.143,-70.819,171.556,28.963,155.396
C06715=1059.232,21.393,-70.835,171.558,28.965,155.396
C06716=1059.239,21.642,-70.850,171.558,28.968,155.397
C06717=1059.245,21.892,-70.866,171.560,28.970,155.397
C06718=1059.251,22.141,-70.881,171.562,28.972,155.397
C06719=1059.257,22.391,-70.897,171.563,28.975,155.398
C06720=1059.264,22.640,-70.912,171.565,28.977,155.398
C06721=1059.269,22.890,-70.928,171.566,28.980,155.398
C06722=1059.275,23.139,-70.943,171.568,28.982,155.399
C06723=1059.281,23.389,-70.959,171.569,28.985,155.399
C06724=1059.288,23.638,-70.974,171.571,28.987,155.399
C06725=1059.294,23.887,-70.991,171.573,28.990,155.400
C06726=1059.300,24.137,-71.006,171.574,28.992,155.400
C06727=1059.306,24.386,-71.022,171.575,28.995,155.400
C06728=1059.312,24.636,-71.037,171.577,28.997,155.401
C06729=1059.318,24.885,-71.053,171.578,28.999,155.401
C06730=1059.325,25.135,-71.068,171.580,29.002,155.401
C06731=1059.331,25.384,-71.084,171.582,29.004,155.402
C06732=1059.336,25.634,-71.100,171.582,29.006,155.402
C06733=1059.343,25.883,-71.115,171.584,29.009,155.402
C06734=1059.349,26.132,-71.132,171.586,29.011,155.403
C06735=1059.355,26.381,-71.146,171.587,29.014,155.403
C06736=1059.361,26.631,-71.163,171.589,29.016,155.403
C06737=1059.367,26.880,-71.178,171.590,29.018,155.404
C06738=1059.373,27.130,-71.194,171.591,29.021,155.404
C06739=1059.379,27.379,-71.210,171.593,29.023,155.404
C06740=1059.385,27.629,-71.225,171.595,29.026,155.405
C06741=1059.391,27.878,-71.241,171.596,29.028,155.405
C06742=1059.398,28.127,-71.257,171.597,29.030,155.405
C06743=1059.403,28.377,-71.272,171.599,29.033,155.406
C06744=1059.409,28.626,-71.289,171.601,29.035,155.406
C06745=1059.416,28.875,-71.304,171.602,29.038,155.406
C06746=1059.422,29.125,-71.320,171.604,29.040,155.407
C06747=1059.428,29.375,-71.336,171.605,29.043,155.407
C06748=1059.435,29.660,-71.354,171.607,29.046,155.407
C06749=1059.442,29.944,-71.372,171.609,29.049,155.408
C06750=1059.449,30.230,-71.391,171.610,29.051,155.408
C06751=1059.455,30.514,-71.409,171.612,29.054,155.409
C06752=1059.461,30.764,-71.424,171.614,29.057,155.409
C06753=1059.467,31.013,-71.441,171.615,29.059,155.409
C06754=1059.473,31.262,-71.457,171.616,29.062,155.410
C06755=1059.479,31.512,-71.473,171.618,29.064,155.410
C06756=1059.486,31.761,-71.488,171.620,29.067,155.410
C06757=1059.492,32.011,-71.504,171.621,29.069,155.411
C06758=1059.498,32.260,-71.521,171.622,29.071,155.411
C06759=1059.504,32.509,-71.537,171.624,29.074,155.412
C06760=1059.510,32.758,-71.552,171.625,29.076,155.412
C06761=1059.516,33.008,-71.568,171.627,29.079,155.412
C06762=1059.522,33.258,-71.584,171.629,29.081,155.412
C06763=1059.528,33.508,-71.601,171.629,29.084,155.413
C06764=1059.534,33.757,-71.617,171.631,29.086,155.413
C06765=1059.541,34.006,-71.633,171.633,29.089,155.414
C06766=1059.547,34.255,-71.649,171.634,29.091,155.414
C06767=1059.553,34.505,-71.665,171.635,29.094,155.414
C06768=1059.559,34.755,-71.681,171.637,29.096,155.415
C06769=1059.565,35.004,-71.697,171.638,29.099,155.415
C06770=1059.571,35.253,-71.713,171.640,29.101,155.415
C06771=1059.577,35.502,-71.729,171.642,29.104,155.416
C06772=1059.583,35.752,-71.745,171.642,29.106,155.416
C06773=1059.589,36.001,-71.762,171.644,29.108,155.416
C06774=1059.595,36.250,-71.778,171.646,29.111,155.417
C06775=1059.602,36.500,-71.793,171.648,29.113,155.417
C06776=1059.608,36.749,-71.810,171.649,29.116,155.417
C06777=1059.614,36.999,-71.826,171.650,29.118,155.418
C06778=1059.620,37.248,-71.843,171.652,29.121,155.418
C06779=1059.626,37.498,-71.859,171.653,29.123,155.418
C06780=1059.633,37.747,-71.875,171.655,29.126,155.419
C06781=1059.638,37.997,-71.890,171.657,29.129,155.419
C06782=1059.644,38.246,-71.906,171.657,29.131,155.419
C06783=1059.650,38.495,-71.923,171.659,29.133,155.420
C06784=1059.656,38.745,-71.939,171.661,29.136,155.420
C06785=1059.663,38.993,-71.956,171.662,29.138,155.421
C06786=1059.669,39.243,-71.972,171.664,29.141,155.421
C06787=1059.675,39.493,-71.989,171.665,29.143,155.421
C06788=1059.681,39.742,-72.005,171.666,29.146,155.422
C06789=1059.687,39.991,-72.021,171.668,29.149,155.422
C06790=1059.693,40.241,-72.037,171.670,29.151,155.422
C06791=1059.699,40.490,-72.054,171.671,29.154,155.423
C06792=1059.705,40.740,-72.070,171.672,29.156,155.423
C06793=1059.711,40.989,-72.086,171.674,29.158,155.423
C06794=1059.716,41.239,-72.103,171.676,29.161,155.424
C06795=1059.722,41.488,-72.119,171.677,29.164,155.424
C06796=1059.728,41.738,-72.136,171.678,29.166,155.424
C06797=1059.734,41.987,-72.152,171.680,29.169,155.425
C06798=1059.741,42.236,-72.169,171.681,29.171,155.425
C06799=1059.747,42.485,-72.185,171.683,29.174,155.426
C06800=1059.753,42.735,-72.202,171.685,29.176,155.426
C06801=1059.759,42.984,-72.218,171.685,29.178,155.426
C06802=1059.765,43.234,-72.235,171.687,29.181,155.427
C06803=1059.771,43.483,-72.251,171.689,29.184,155.427
C06804=1059.777,43.733,-72.267,171.690,29.186,155.427
C06805=1059.783,43.982,-72.284,171.692,29.189,155.428
C06806=1059.789,44.231,-72.300,171.693,29.191,155.428
C06807=1059.794,44.481,-72.317,171.694,29.194,155.428
C06808=1059.800,44.730,-72.333,171.696,29.196,155.429
C06809=1059.807,44.980,-72.350,171.698,29.199,155.429
C06810=1059.813,45.229,-72.367,171.698,29.202,155.430
C06811=1059.818,45.478,-72.384,171.700,29.204,155.430
C06812=1059.825,45.763,-72.403,171.702,29.207,155.430
C06813=1059.832,46.047,-72.421,171.703,29.210,155.431
C06814=1059.839,46.332,-72.440,171.705,29.213,155.431
C06815=1059.845,46.618,-72.460,171.707,29.216,155.432
C06816=1059.851,46.867,-72.476,171.708,29.218,155.432
C06817=1059.857,47.116,-72.493,171.710,29.221,155.432
C06818=1059.864,47.365,-72.510,171.712,29.224,155.433
C06819=1059.869,47.615,-72.527,171.712,29.226,155.433
C06820=1059.875,47.865,-72.543,171.714,29.229,155.434
C06821=1059.882,48.113,-72.560,171.716,29.231,155.434
C06822=1059.887,48.363,-72.577,171.717,29.234,155.434
C06823=1059.893,48.612,-72.593,171.719,29.236,155.435
C06824=1059.900,48.862,-72.610,171.720,29.239,155.435
C06825=1059.906,49.111,-72.627,171.722,29.242,155.435
C06826=1059.911,49.361,-72.644,171.723,29.244,155.436
C06827=1059.917,49.610,-72.661,171.725,29.246,155.436
C06828=1059.923,49.859,-72.677,171.726,29.249,155.437
C06829=1059.929,50.109,-72.694,171.727,29.252,155.437
C06830=1059.935,50.358,-72.711,171.729,29.255,155.437
C06831=1059.941,50.607,-72.727,171.731,29.257,155.438
C06832=1059.947,50.856,-72.744,171.732,29.260,155.438
C06833=1059.953,51.106,-72.761,171.733,29.262,155.438
C06834=1059.959,51.355,-72.778,171.735,29.264,155.439
C06835=1059.965,51.605,-72.795,171.736,29.267,155.439
C06836=1059.971,51.854,-72.811,171.738,29.270,155.439
C06837=1059.977,52.104,-72.829,171.739,29.272,155.440
C06838=1059.983,52.353,-72.845,171.740,29.274,155.440
C06839=1059.989,52.602,-72.863,171.742,29.277,155.441
C06840=1059.995,52.851,-72.879,171.744,29.280,155.441
C06841=1060.002,53.101,-72.896,171.746,29.282,155.441
C06842=1060.007,53.350,-72.913,171.746,29.285,155.442
C06843=1060.013,53.599,-72.930,171.748,29.288,155.442
C06844=1060.020,53.849,-72.947,171.750,29.290,155.442
C06845=1060.025,54.098,-72.964,171.751,29.292,155.443
C06846=1060.031,54.348,-72.980,171.753,29.295,155.443
C06847=1060.038,54.597,-72.998,171.754,29.298,155.444
C06848=1060.043,54.847,-73.015,171.755,29.300,155.444
C06849=1060.050,55.095,-73.032,171.757,29.303,155.444
C06850=1060.056,55.346,-73.048,171.759,29.305,155.445
C06851=1060.062,55.595,-73.066,171.759,29.307,155.445
C06852=1060.068,55.844,-73.082,171.761,29.310,155.445
C06853=1060.074,56.093,-73.099,171.763,29.313,155.446
C06854=1060.080,56.342,-73.117,171.764,29.316,155.446
C06855=1060.086,56.592,-73.133,171.766,29.318,155.446
C06856=1060.093,56.841,-73.151,171.767,29.320,155.447
C06857=1060.098,57.091,-73.167,171.769,29.323,155.447
C06858=1060.104,57.340,-73.184,171.770,29.325,155.448
C06859=1060.110,57.589,-73.202,171.772,29.328,155.448
C06860=1060.116,57.839,-73.219,171.774,29.331,155.448
C06861=1060.123,58.087,-73.236,171.774,29.333,155.449
C06862=1060.128,58.338,-73.253,171.776,29.336,155.449
C06863=1060.135,58.586,-73.270,171.778,29.338,155.449
C06864=1060.141,58.836,-73.287,171.779,29.341,155.450
C06865=1060.147,59.086,-73.304,171.780,29.343,155.450
C06866=1060.153,59.334,-73.321,171.782,29.346,155.451
C06867=1060.159,59.584,-73.339,171.784,29.348,155.451
C06868=1060.165,59.833,-73.355,171.785,29.351,155.451
C06869=1060.172,60.083,-73.372,171.787,29.354,155.452
C06870=1060.177,60.332,-73.390,171.788,29.355,155.452
C06871=1060.184,60.581,-73.407,171.789,29.358,155.452
C06872=1060.189,60.831,-73.424,171.791,29.361,155.453
C06873=1060.196,61.080,-73.441,171.793,29.363,155.453
C06874=1060.203,61.329,-73.459,171.794,29.366,155.453
C06875=1060.208,61.579,-73.475,171.795,29.368,155.454
C06876=1060.215,61.863,-73.495,171.797,29.371,155.454
C06877=1060.223,62.147,-73.515,171.798,29.374,155.455
C06878=1060.229,62.433,-73.534,171.800,29.377,155.455
C06879=1060.236,62.717,-73.554,171.802,29.379,155.455
C06880=1060.242,62.967,-73.572,171.803,29.382,155.456
C06881=1060.249,63.215,-73.589,171.805,29.385,155.456
C06882=1060.256,63.465,-73.606,171.807,29.387,155.456
C06883=1060.261,63.714,-73.623,171.809,29.390,155.457
C06884=1060.267,63.963,-73.640,171.809,29.392,155.457
C06885=1060.273,64.213,-73.658,171.811,29.395,155.458
C06886=1060.279,64.462,-73.675,171.813,29.397,155.458
C06887=1060.286,64.711,-73.693,171.814,29.400,155.458
C06888=1060.291,64.960,-73.711,171.816,29.403,155.459
C06889=1060.298,65.210,-73.727,171.817,29.405,155.459
C06890=1060.303,65.459,-73.745,171.818,29.408,155.460
C06891=1060.310,65.709,-73.762,171.820,29.410,155.460
C06892=1060.316,65.958,-73.780,171.822,29.413,155.460
C06893=1060.322,66.208,-73.798,171.824,29.415,155.461
C06894=1060.328,66.456,-73.815,171.824,29.418,155.461
C06895=1060.334,66.706,-73.832,171.826,29.421,155.461
C06896=1060.340,66.955,-73.850,171.828,29.423,155.462
C06897=1060.346,67.205,-73.867,171.829,29.425,155.462
C06898=1060.352,67.454,-73.885,171.830,29.428,155.463
C06899=1060.357,67.703,-73.903,171.832,29.431,155.463
C06900=1060.364,67.952,-73.920,171.833,29.434,155.463
C06901=1060.370,68.202,-73.937,171.835,29.436,155.464
C06902=1060.376,68.451,-73.955,171.837,29.438,155.464
C06903=1060.381,68.701,-73.972,171.838,29.441,155.464
C06904=1060.388,68.950,-73.990,171.839,29.444,155.465
C06905=1060.394,69.199,-74.007,171.841,29.446,155.465
C06906=1060.400,69.449,-74.025,171.843,29.449,155.466
C06907=1060.405,69.698,-74.043,171.844,29.451,155.466
C06908=1060.412,69.947,-74.060,171.845,29.454,155.466
C06909=1060.418,70.196,-74.078,171.847,29.457,155.467
C06910=1060.424,70.445,-74.096,171.848,29.459,155.467
C06911=1060.429,70.694,-74.114,171.850,29.462,155.468
C06912=1060.436,70.944,-74.132,171.851,29.464,155.468
C06913=1060.442,71.194,-74.149,171.853,29.467,155.468
C06914=1060.448,71.443,-74.167,171.854,29.470,155.469
C06915=1060.454,71.692,-74.185,171.856,29.472,155.469
C06916=1060.460,71.941,-74.202,171.858,29.475,155.469
C06917=1060.466,72.191,-74.220,171.858,29.477,155.470
C06918=1060.471,72.440,-74.238,171.860,29.480,155.470
C06919=1060.477,72.690,-74.256,171.862,29.483,155.471
C06920=1060.484,72.938,-74.273,171.863,29.485,155.471
C06921=1060.490,73.188,-74.291,171.864,29.488,155.471
C06922=1060.496,73.437,-74.309,171.866,29.491,155.472
C06923=1060.502,73.687,-74.327,171.868,29.493,155.472
C06924=1060.507,73.936,-74.344,171.869,29.495,155.472
C06925=1060.513,74.185,-74.362,171.871,29.498,155.473
C06926=1060.519,74.435,-74.380,171.872,29.501,155.473
C06927=1060.525,74.683,-74.398,171.873,29.504,155.474
C06928=1060.532,74.933,-74.416,171.875,29.506,155.474
C06929=1060.538,75.182,-74.433,171.877,29.508,155.474
C06930=1060.544,75.432,-74.451,171.878,29.511,155.475
C06931=1060.549,75.681,-74.469,171.879,29.514,155.475
C06932=1060.556,75.930,-74.487,171.881,29.516,155.476
C06933=1060.562,76.180,-74.505,171.883,29.519,155.476
C06934=1060.567,76.429,-74.523,171.884,29.521,155.476
C06935=1060.573,76.678,-74.541,171.886,29.524,155.477
C06936=1060.579,76.927,-74.559,171.887,29.527,155.477
C06937=1060.585,77.177,-74.577,171.888,29.529,155.478
C06938=1060.592,77.426,-74.595,171.890,29.532,155.478
C06939=1060.598,77.675,-74.612,171.892,29.534,155.478
C06940=1060.605,77.959,-74.633,171.893,29.538,155.479
C06941=1060.611,78.244,-74.653,171.895,29.540,155.479
C06942=1060.618,78.528,-74.674,171.897,29.543,155.480
C06943=1060.626,78.813,-74.695,171.898,29.546,155.480
C06944=1060.631,79.062,-74.713,171.900,29.549,155.480
C06945=1060.637,79.311,-74.732,171.901,29.551,155.481
C06946=1060.642,79.560,-74.749,171.903,29.554,155.481
C06947=1060.649,79.810,-74.767,171.904,29.557,155.482
C06948=1060.655,80.059,-74.786,171.906,29.559,155.482
C06949=1060.661,80.308,-74.803,171.908,29.562,155.482
C06950=1060.667,80.558,-74.821,171.908,29.565,155.483
C06951=1060.672,80.806,-74.840,171.910,29.567,155.483
C06952=1060.678,81.056,-74.858,171.912,29.570,155.484
C06953=1060.684,81.306,-74.877,171.913,29.573,155.484
C06954=1060.690,81.555,-74.894,171.915,29.576,155.484
C06955=1060.696,81.804,-74.912,171.916,29.577,155.485
C06956=1060.702,82.053,-74.931,171.918,29.580,155.485
C06957=1060.708,82.303,-74.949,171.919,29.583,155.486
C06958=1060.714,82.552,-74.967,171.921,29.586,155.486
C06959=1060.720,82.802,-74.986,171.923,29.588,155.486
C06960=1060.725,83.050,-75.004,171.923,29.591,155.487
C06961=1060.732,83.300,-75.022,171.925,29.594,155.487
C06962=1060.738,83.549,-75.041,171.927,29.596,155.488
C06963=1060.744,83.798,-75.058,171.928,29.599,155.488
C06964=1060.750,84.047,-75.077,171.930,29.601,155.488
C06965=1060.755,84.297,-75.095,171.931,29.604,155.489
C06966=1060.761,84.546,-75.114,171.933,29.607,155.489
C06967=1060.767,84.795,-75.132,171.934,29.609,155.489
C06968=1060.774,85.044,-75.150,171.936,29.612,155.490
C06969=1060.779,85.294,-75.168,171.938,29.615,155.490
C06970=1060.786,85.543,-75.186,171.938,29.617,155.491
C06971=1060.791,85.793,-75.205,171.940,29.619,155.491
C06972=1060.797,86.042,-75.224,171.942,29.622,155.491
C06973=1060.803,86.290,-75.242,171.943,29.625,155.492
C06974=1060.809,86.540,-75.260,171.945,29.628,155.492
C06975=1060.816,86.789,-75.278,171.946,29.630,155.493
C06976=1060.821,87.038,-75.297,171.948,29.632,155.493
C06977=1060.827,87.288,-75.315,171.949,29.635,155.493
C06978=1060.833,87.537,-75.334,171.951,29.638,155.494
C06979=1060.840,87.786,-75.352,171.953,29.641,155.494
C06980=1060.846,88.036,-75.371,171.953,29.643,155.495
C06981=1060.851,88.285,-75.389,171.955,29.646,155.495
C06982=1060.857,88.534,-75.407,171.957,29.648,155.495
C06983=1060.864,88.783,-75.426,171.959,29.651,155.496
C06984=1060.870,89.033,-75.444,171.960,29.653,155.496
C06985=1060.876,89.281,-75.462,171.962,29.656,155.496
C06986=1060.881,89.531,-75.481,171.963,29.659,155.497
C06987=1060.887,89.781,-75.499,171.965,29.661,155.497
C06988=1060.894,90.030,-75.518,171.966,29.664,155.498
C06989=1060.900,90.279,-75.537,171.968,29.666,155.498
C06990=1060.905,90.527,-75.556,171.970,29.669,155.498
C06991=1060.911,90.777,-75.573,171.970,29.672,155.499
C06992=1060.918,91.026,-75.592,171.972,29.674,155.499
C06993=1060.924,91.276,-75.611,171.974,29.677,155.500
C06994=1060.929,91.524,-75.630,171.975,29.680,155.500
C06995=1060.935,91.774,-75.648,171.977,29.682,155.500
C06996=1060.941,92.023,-75.667,171.978,29.684,155.501
C06997=1060.947,92.273,-75.686,171.980,29.687,155.501
C06998=1060.953,92.521,-75.704,171.981,29.690,155.502
C06999=1060.959,92.771,-75.722,171.983,29.693,155.502
C07000=1060.965,93.020,-75.742,171.985,29.695,155.502
C07001=1060.971,93.270,-75.760,171.985,29.698,155.503
C07002=1060.977,93.519,-75.779,171.987,29.701,155.503
C07003=1060.982,93.767,-75.798,171.989,29.703,155.504
C07004=1060.989,94.052,-75.820,171.991,29.706,155.504
C07005=1060.996,94.336,-75.841,171.992,29.709,155.504
C07006=1061.003,94.621,-75.862,171.994,29.712,155.505
C07007=1061.010,94.905,-75.884,171.996,29.715,155.505
C07008=1061.015,95.155,-75.902,171.997,29.718,155.506
C07009=1061.021,95.404,-75.921,171.999,29.721,155.506
C07010=1061.027,95.653,-75.940,172.001,29.723,155.507
C07011=1061.033,95.902,-75.958,172.002,29.726,155.507
C07012=1061.039,96.152,-75.978,172.004,29.728,155.507
C07013=1061.046,96.401,-75.996,172.005,29.731,155.508
C07014=1061.051,96.650,-76.016,172.007,29.734,155.508
C07015=1061.057,96.899,-76.034,172.008,29.736,155.509
C07016=1061.063,97.148,-76.053,172.010,29.739,155.509
C07017=1061.069,97.397,-76.072,172.012,29.742,155.509
C07018=1061.075,97.647,-76.091,172.012,29.744,155.510
C07019=1061.081,97.896,-76.110,172.014,29.747,155.510
C07020=1061.087,98.145,-76.129,172.016,29.749,155.510
C07021=1061.093,98.394,-76.148,172.018,29.752,155.511
C07022=1061.099,98.644,-76.167,172.019,29.755,155.511
C07023=1061.106,98.893,-76.185,172.021,29.757,155.512
C07024=1061.111,99.142,-76.204,172.022,29.760,155.512
C07025=1061.117,99.391,-76.223,172.023,29.763,155.513
C07026=1061.123,99.640,-76.242,172.025,29.765,155.513
C07027=1061.129,99.889,-76.261,172.027,29.768,155.513
C07028=1061.135,100.139,-76.280,172.029,29.770,155.514
C07029=1061.141,100.388,-76.299,172.030,29.773,155.514
C07030=1061.147,100.637,-76.318,172.031,29.775,155.514
C07031=1061.153,100.887,-76.337,172.033,29.778,155.515
C07032=1061.159,101.136,-76.356,172.034,29.781,155.515
C07033=1061.165,101.385,-76.375,172.036,29.784,155.516
C07034=1061.170,101.635,-76.394,172.038,29.786,155.516
C07035=1061.176,101.883,-76.413,172.040,29.789,155.516
C07036=1061.182,102.133,-76.432,172.040,29.792,155.517
C07037=1061.188,102.382,-76.451,172.042,29.794,155.517
C07038=1061.194,102.631,-76.471,172.044,29.797,155.518
C07039=1061.200,102.880,-76.490,172.045,29.800,155.518
C07040=1061.206,103.129,-76.509,172.047,29.802,155.519
C07041=1061.211,103.379,-76.528,172.049,29.805,155.519
C07042=1061.217,103.628,-76.547,172.051,29.808,155.519
C07043=1061.224,103.877,-76.566,172.051,29.810,155.520
C07044=1061.230,104.126,-76.586,172.053,29.813,155.520
C07045=1061.235,104.376,-76.605,172.055,29.815,155.520
C07046=1061.241,104.625,-76.625,172.057,29.818,155.521
C07047=1061.247,104.874,-76.644,172.058,29.821,155.521
C07048=1061.253,105.122,-76.663,172.060,29.823,155.522
C07049=1061.258,105.372,-76.682,172.061,29.826,155.522
C07050=1061.264,105.621,-76.701,172.062,29.829,155.523
C07051=1061.270,105.871,-76.720,172.064,29.831,155.523
C07052=1061.277,106.119,-76.740,172.066,29.834,155.523
C07053=1061.282,106.369,-76.759,172.068,29.837,155.524
C07054=1061.288,106.618,-76.778,172.069,29.840,155.524
C07055=1061.294,106.867,-76.798,172.071,29.842,155.525
C07056=1061.300,107.116,-76.818,172.072,29.845,155.525
C07057=1061.306,107.365,-76.836,172.073,29.847,155.525
C07058=1061.312,107.615,-76.855,172.075,29.850,155.526
C07059=1061.318,107.864,-76.875,172.077,29.852,155.526
C07060=1061.323,108.113,-76.895,172.079,29.855,155.526
C07061=1061.329,108.362,-76.914,172.080,29.858,155.527
C07062=1061.336,108.611,-76.933,172.081,29.860,155.527
C07063=1061.341,108.860,-76.952,172.083,29.863,155.528
C07064=1061.347,109.110,-76.972,172.085,29.866,155.528
C07065=1061.353,109.359,-76.992,172.086,29.868,155.529
C07066=1061.359,109.608,-77.011,172.088,29.871,155.529
C07067=1061.366,109.858,-77.030,172.090,29.874,155.529
C07068=1061.372,110.142,-77.052,172.091,29.877,155.530
C07069=1061.379,110.427,-77.074,172.093,29.880,155.530
C07070=1061.386,110.711,-77.097,172.095,29.883,155.531
C07071=1061.393,110.995,-77.119,172.096,29.886,155.531
C07072=1061.399,111.244,-77.139,172.098,29.888,155.531
C07073=1061.404,111.493,-77.158,172.100,29.891,155.532
C07074=1061.410,111.742,-77.178,172.102,29.893,155.532
C07075=1061.416,111.992,-77.197,172.103,29.896,155.533
C07076=1061.422,112.240,-77.217,172.105,29.899,155.533
C07077=1061.428,112.491,-77.237,172.107,29.902,155.534
C07078=1061.434,112.739,-77.256,172.108,29.904,155.534
C07079=1061.440,112.989,-77.276,172.109,29.907,155.534
C07080=1061.446,113.238,-77.296,172.111,29.909,155.535
C07081=1061.452,113.487,-77.315,172.113,29.912,155.535
C07082=1061.458,113.736,-77.335,172.114,29.915,155.536
C07083=1061.463,113.985,-77.354,172.116,29.918,155.536
C07084=1061.469,114.234,-77.374,172.118,29.920,155.536
C07085=1061.475,114.484,-77.393,172.120,29.923,155.537
C07086=1061.481,114.732,-77.413,172.120,29.926,155.537
C07087=1061.487,114.982,-77.433,172.122,29.928,155.538
C07088=1061.493,115.231,-77.453,172.124,29.931,155.538
C07089=1061.498,115.480,-77.473,172.125,29.934,155.538
C07090=1061.504,115.729,-77.492,172.127,29.936,155.539
C07091=1061.510,115.978,-77.512,172.129,29.939,155.539
C07092=1061.516,116.227,-77.532,172.131,29.942,155.540
C07093=1061.521,116.476,-77.551,172.131,29.945,155.540
C07094=1061.527,116.726,-77.572,172.133,29.948,155.541
C07095=1061.533,116.976,-77.592,172.135,29.950,155.541
C07096=1061.539,117.224,-77.612,172.137,29.953,155.541
C07097=1061.545,117.473,-77.632,172.138,29.956,155.542
C07098=1061.551,117.722,-77.652,172.140,29.958,155.542
C07099=1061.556,117.972,-77.671,172.142,29.961,155.543
C07100=1061.562,118.221,-77.691,172.143,29.964,155.543
C07101=1061.568,118.469,-77.711,172.145,29.967,155.543
C07102=1061.573,118.719,-77.731,172.146,29.969,155.544
C07103=1061.579,118.968,-77.750,172.148,29.972,155.544
C07104=1061.585,119.217,-77.771,172.149,29.974,155.545
C07105=1061.591,119.467,-77.791,172.151,29.977,155.545
C07106=1061.597,119.716,-77.811,172.153,29.980,155.546
C07107=1061.603,119.964,-77.831,172.155,29.983,155.546
C07108=1061.608,120.214,-77.851,172.156,29.985,155.546
C07109=1061.614,120.462,-77.871,172.158,29.988,155.547
C07110=1061.620,120.712,-77.890,172.160,29.991,155.547
C07111=1061.627,120.961,-77.911,172.160,29.993,155.548
C07112=1061.632,121.210,-77.931,172.162,29.996,155.548
C07113=1061.638,121.459,-77.951,172.164,29.999,155.548
C07114=1061.644,121.708,-77.971,172.166,30.001,155.549
C07115=1061.649,121.958,-77.990,172.167,30.004,155.549
C07116=1061.655,122.207,-78.011,172.169,30.007,155.550
C07117=1061.661,122.456,-78.031,172.171,30.009,155.550
C07118=1061.667,122.705,-78.051,172.173,30.012,155.550
C07119=1061.673,122.954,-78.071,172.174,30.015,155.551
C07120=1061.679,123.203,-78.092,172.176,30.017,155.551
C07121=1061.684,123.452,-78.111,172.178,30.020,155.552
C07122=1061.691,123.702,-78.131,172.178,30.023,155.552
C07123=1061.697,123.951,-78.151,172.180,30.025,155.553
C07124=1061.702,124.200,-78.172,172.182,30.028,155.553
C07125=1061.708,124.449,-78.192,172.184,30.031,155.553
C07126=1061.715,124.698,-78.212,172.185,30.033,155.554
C07127=1061.721,124.947,-78.232,172.187,30.036,155.554
C07128=1061.726,125.196,-78.253,172.189,30.039,155.555
C07129=1061.732,125.445,-78.273,172.191,30.042,155.555
C07130=1061.739,125.694,-78.293,172.192,30.044,155.555
C07131=1061.744,125.944,-78.313,172.194,30.047,155.556
C07132=1061.751,126.228,-78.336,172.196,30.050,155.556
C07133=1061.757,126.513,-78.359,172.197,30.053,155.557
C07134=1061.764,126.796,-78.382,172.199,30.056,155.557
C07135=1061.770,127.081,-78.405,172.202,30.059,155.558
C07136=1061.777,127.330,-78.425,172.203,30.062,155.558
C07137=1061.783,127.579,-78.445,172.204,30.064,155.558
C07138=1061.789,127.828,-78.465,172.206,30.067,155.559
C07139=1061.795,128.077,-78.487,172.208,30.070,155.559
C07140=1061.801,128.326,-78.507,172.210,30.072,155.560
C07141=1061.807,128.575,-78.527,172.211,30.075,155.560
C07142=1061.812,128.824,-78.547,172.213,30.078,155.561
C07143=1061.819,129.073,-78.568,172.215,30.080,155.561
C07144=1061.825,129.322,-78.588,172.216,30.083,155.561
C07145=1061.830,129.571,-78.608,172.218,30.086,155.562
C07146=1061.837,129.821,-78.629,172.220,30.088,155.562
C07147=1061.843,130.070,-78.648,172.222,30.091,155.562
C07148=1061.849,130.320,-78.669,172.223,30.093,155.563
C07149=1061.855,130.568,-78.689,172.225,30.096,155.563
C07150=1061.861,130.817,-78.709,172.227,30.099,155.564
C07151=1061.867,131.066,-78.731,172.229,30.101,155.564
C07152=1061.873,131.315,-78.751,172.230,30.104,155.565
C07153=1061.879,131.564,-78.771,172.232,30.107,155.565
C07154=1061.885,131.814,-78.792,172.233,30.109,155.565
C07155=1061.891,132.063,-78.812,172.235,30.112,155.566
C07156=1061.896,132.312,-78.832,172.236,30.115,155.566
C07157=1061.902,132.561,-78.854,172.238,30.117,155.567
C07158=1061.908,132.810,-78.874,172.240,30.120,155.567
C07159=1061.913,133.059,-78.894,172.242,30.123,155.567
C07160=1061.920,133.308,-78.915,172.243,30.125,155.568
C07161=1061.925,133.557,-78.936,172.245,30.128,155.568
C07162=1061.931,133.806,-78.957,172.247,30.131,155.569
C07163=1061.937,134.056,-78.977,172.249,30.134,155.569
C07164=1061.943,134.305,-78.997,172.250,30.137,155.570
C07165=1061.949,134.553,-79.018,172.252,30.140,155.570
C07166=1061.955,134.803,-79.039,172.254,30.142,155.570
C07167=1061.960,135.052,-79.060,172.255,30.145,155.571
C07168=1061.966,135.300,-79.080,172.257,30.148,155.571
C07169=1061.972,135.550,-79.101,172.259,30.150,155.572
C07170=1061.978,135.799,-79.121,172.261,30.153,155.572
C07171=1061.984,136.048,-79.143,172.262,30.156,155.572
C07172=1061.989,136.297,-79.163,172.264,30.158,155.573
C07173=1061.995,136.546,-79.183,172.266,30.161,155.573
C07174=1062.002,136.795,-79.205,172.268,30.164,155.574
C07175=1062.007,137.044,-79.226,172.269,30.166,155.574
C07176=1062.013,137.294,-79.246,172.271,30.169,155.574
C07177=1062.019,137.542,-79.267,172.273,30.172,155.575
C07178=1062.024,137.791,-79.288,172.275,30.174,155.575
C07179=1062.031,138.040,-79.309,172.276,30.177,155.576
C07180=1062.036,138.289,-79.329,172.278,30.180,155.576
C07181=1062.042,138.539,-79.350,172.280,30.182,155.577
C07182=1062.049,138.787,-79.371,172.282,30.185,155.577
C07183=1062.054,139.037,-79.392,172.282,30.188,155.577
C07184=1062.060,139.286,-79.413,172.284,30.190,155.578
C07185=1062.066,139.534,-79.433,172.286,30.194,155.578
C07186=1062.072,139.784,-79.455,172.288,30.196,155.579
C07187=1062.077,140.033,-79.475,172.289,30.199,155.579
C07188=1062.084,140.282,-79.497,172.291,30.202,155.580
C07189=1062.089,140.531,-79.517,172.293,30.204,155.580
C07190=1062.096,140.780,-79.538,172.295,30.207,155.580
C07191=1062.101,141.029,-79.559,172.296,30.210,155.581
C07192=1062.107,141.278,-79.581,172.298,30.212,155.581
C07193=1062.112,141.528,-79.601,172.300,30.215,155.582
C07194=1062.118,141.776,-79.622,172.302,30.218,155.582
C07195=1062.124,142.026,-79.643,172.303,30.221,155.583
C07196=1062.131,142.310,-79.667,172.306,30.224,155.583
C07197=1062.137,142.594,-79.691,172.308,30.227,155.583
C07198=1062.144,142.878,-79.715,172.309,30.230,155.584
C07199=1062.151,143.162,-79.739,172.312,30.233,155.584
C07200=1062.157,143.411,-79.761,172.314,30.236,155.585
C07201=1062.162,143.660,-79.782,172.316,30.239,155.585
C07202=1062.168,143.910,-79.803,172.317,30.242,155.586
C07203=1062.174,144.158,-79.824,172.319,30.245,155.586
C07204=1062.180,144.408,-79.845,172.321,30.247,155.587
C07205=1062.186,144.656,-79.866,172.323,30.250,155.587
C07206=1062.192,144.905,-79.888,172.324,30.253,155.587
C07207=1062.197,145.154,-79.908,172.326,30.255,155.588
C07208=1062.204,145.404,-79.930,172.328,30.258,155.588
C07209=1062.209,145.652,-79.951,172.330,30.261,155.589
C07210=1062.215,145.902,-79.972,172.331,30.263,155.589
C07211=1062.221,146.150,-79.993,172.333,30.266,155.589
C07212=1062.227,146.400,-80.015,172.335,30.269,155.590
C07213=1062.232,146.648,-80.036,172.337,30.272,155.590
C07214=1062.239,146.898,-80.057,172.338,30.275,155.591
C07215=1062.245,147.147,-80.078,172.340,30.277,155.591
C07216=1062.251,147.395,-80.099,172.342,30.280,155.592
C07217=1062.257,147.645,-80.121,172.344,30.283,155.592
C07218=1062.262,147.894,-80.142,172.345,30.285,155.592
C07219=1062.268,148.143,-80.163,172.347,30.288,155.593
C07220=1062.274,148.391,-80.185,172.349,30.291,155.593
C07221=1062.280,148.641,-80.206,172.351,30.293,155.594
C07222=1062.286,148.889,-80.227,172.352,30.297,155.594
C07223=1062.291,149.139,-80.248,172.354,30.299,155.595
C07224=1062.298,149.388,-80.270,172.356,30.302,155.595
C07225=1062.303,149.637,-80.291,172.358,30.305,155.595
C07226=1062.309,149.886,-80.314,172.359,30.307,155.596
C07227=1062.314,150.135,-80.335,172.361,30.310,155.596
C07228=1062.320,150.384,-80.356,172.363,30.313,155.597
C07229=1062.326,150.633,-80.378,172.364,30.316,155.597
C07230=1062.332,150.882,-80.399,172.366,30.319,155.598
C07231=1062.338,151.131,-80.421,172.368,30.321,155.598
C07232=1062.343,151.380,-80.442,172.371,30.324,155.598
C07233=1062.350,151.629,-80.463,172.372,30.327,155.599
C07234=1062.355,151.878,-80.484,172.374,30.329,155.599
C07235=1062.361,152.127,-80.507,172.376,30.333,155.600
C07236=1062.367,152.376,-80.528,172.378,30.335,155.600
C07237=1062.372,152.625,-80.550,172.379,30.338,155.601
C07238=1062.378,152.874,-80.571,172.381,30.341,155.601
C07239=1062.385,153.123,-80.593,172.383,30.343,155.601
C07240=1062.390,153.372,-80.614,172.385,30.346,155.602
C07241=1062.396,153.621,-80.636,172.386,30.349,155.602
C07242=1062.402,153.871,-80.658,172.388,30.352,155.603
C07243=1062.407,154.119,-80.679,172.390,30.355,155.603
C07244=1062.413,154.368,-80.701,172.392,30.357,155.604
C07245=1062.419,154.617,-80.722,172.393,30.360,155.604
C07246=1062.425,154.866,-80.744,172.395,30.363,155.604
C07247=1062.431,155.115,-80.765,172.398,30.366,155.605
C07248=1062.436,155.363,-80.788,172.400,30.369,155.605
C07249=1062.443,155.613,-80.810,172.401,30.371,155.606
C07250=1062.449,155.862,-80.831,172.403,30.374,155.606
C07251=1062.454,156.111,-80.853,172.405,30.377,155.607
C07252=1062.460,156.360,-80.875,172.407,30.379,155.607
C07253=1062.466,156.609,-80.896,172.408,30.383,155.608
C07254=1062.472,156.857,-80.918,172.410,30.385,155.608
C07255=1062.477,157.107,-80.940,172.412,30.388,155.608
C07256=1062.483,157.356,-80.962,172.414,30.391,155.609
C07257=1062.490,157.605,-80.984,172.416,30.393,155.609
C07258=1062.494,157.854,-81.006,172.417,30.397,155.610
C07259=1062.501,158.103,-81.027,172.420,30.399,155.610
C07260=1062.508,158.386,-81.052,172.422,30.403,155.611
C07261=1062.514,158.670,-81.077,172.423,30.405,155.611
C07262=1062.520,158.955,-81.102,172.426,30.409,155.612
C07263=1062.527,159.239,-81.127,172.428,30.412,155.612
C07264=1062.533,159.487,-81.148,172.430,30.415,155.613
C07265=1062.539,159.736,-81.171,172.431,30.417,155.613
C07266=1062.545,159.985,-81.193,172.433,30.421,155.613
C07267=1062.551,160.234,-81.215,172.436,30.423,155.614
C07268=1062.556,160.483,-81.236,172.438,30.426,155.614
C07269=1062.562,160.732,-81.259,172.439,30.429,155.615
